// ---- POUs/AFL extensions/analog_actuator/commands/analog_actuator_deactivate.TcPOU
(*$
	Sends a deactivation command to the instance <b><i>this</i></b>, i.e.
	requests the instance to deactivate the linked <a href="#digital_output_object"><i>digital_output</i></a> <br/>	
	to reach the status <a href="#analog_actuator_status_enum"><i>ANALOG_ACTUATOR_STATUS_INACTIVE</i></a>
	The command is accepted only in <a href="#mode_enum"><i>MODE_OPERATIONAL</i></a>, the object is not faulted
	and the fault reaction is <a href="#analog_actuator_fault_reaction_enum"><i>ANALOG_ACTUATOR_FAULT_REACTION_IGNORE</i></a>.<br/>
	The method returns <i>TRUE</i> if the command is accepted, otherwise it returns <i>FALSE</i>.
$*)
FUNCTION analog_actuator_deactivate : BOOL
VAR_IN_OUT
    CONVERSION_this:	analog_actuator;	(*$ Instance to which the method applies $*)
END_VAR

IF	NOT (descriptor_mode_is_operational(CONVERSION_this.descriptor)
		OR
		descriptor_mode_is_test(CONVERSION_this.descriptor))
	OR	(
			(	descriptor_is_not_ready(CONVERSION_this.descriptor)
				AND
				CONVERSION_this.fault_reaction <> ANALOG_ACTUATOR_FAULT_REACTION_IGNORE	)
		)
THEN
	analog_actuator_deactivate := FALSE;					(* command rejected *)
 	RETURN;
END_IF

CONVERSION_this.operational_command := ANALOG_ACTUATOR_CMD_DEACTIVATE;
CONVERSION_this.analog_physical_command := 0;
analog_actuator_deactivate := TRUE;						(* command accepted *)

END_FUNCTION

// ---- POUs/AFL extensions/analog_actuator/commands/analog_actuator_set_feedback_tolerance.TcPOU
(*$
	Set Lower and Upper Feedback tolerance to the instance <b><i>this</i></b>,
	The command is accepted only in <a href="#mode_enum"><i>MODE_OPERATIONAL</i></a>
	and analog_actuator_add_ai_feedback has been called at startup
	The method returns <i>TRUE</i> if the command is accepted, otherwise it returns <i>FALSE</i>.
$*)
FUNCTION analog_actuator_set_feedback_tolerance : BOOL
VAR_INPUT
	feedback_upper_tolerance:		REAL;			(*$ Upper Tolerance Physical Value $*)
	feedback_lower_tolerance:		REAL;			(*$ Lower Tolerance Physical Value $*)
END_VAR
VAR_IN_OUT
    CONVERSION_this:	analog_actuator;	(*$ Instance to which the method applies $*)
END_VAR

IF	NOT (descriptor_mode_is_operational(CONVERSION_this.descriptor)
		OR
		descriptor_mode_is_test(CONVERSION_this.descriptor))
	OR
	NOT CONVERSION_this.has_ai_feedback
THEN
	analog_actuator_set_feedback_tolerance := FALSE;					(* command rejected *)
 	RETURN;
END_IF

CONVERSION_this.feedback_lower_tolerance := feedback_lower_tolerance;
CONVERSION_this.feedback_upper_tolerance := feedback_upper_tolerance;

analog_actuator_set_feedback_tolerance := TRUE;						(* command accepted *)

END_FUNCTION

// ---- POUs/AFL extensions/analog_actuator/initialize/analog_actuator_add_ai_feedback.TcPOU
(*$
	The method adds the <a href="#analog_input_object"><i>analog_input</i></a> that performs 
	the active feedback to the instance specified by the parameter <i><b>this</b></i>.<br/>
	<p>
	This function should be called at startup only.<br/>	
	Against errors on the input parameters the cpu is stopped, in this case the cause <br/>
	can be inspected in the global struct <i>framework.abort_error</i>: <br/>
	<br/>
	<ul>
    <li> ERRORID_1 = 9: <b><i>this</i></b> instance has already an active digital_input </li>
    <li> ERRORID_1 = 12: <b><i>this</i></b> instance is a real value check type </li>
	</ul>
	</p>
$*)
FUNCTION analog_actuator_add_ai_feedback : VOID
VAR_INPUT
	achk_diagnosis_max_value:		REAL;
	(*$ Value over which auto-diagnosis message is triggered; $*)
	achk_diagnosis_min_value:		REAL;
	(*$ Value under which auto-diagnosis message is triggered; $*)
	achk_offset:					REAL;
	(*$ Offset added (subtracted if polarity_direct is FALSE) to the other limits.
		Ex. if offset = 0 and max_value =100, out_of_upper_range is triggered if value>100
		if offset = 10 and max_value =100, out_of_upper_range is triggered if value>110 $*)
	achk_hysteresis:				UDINT;
	(*$ Hysteresis on max or min value. If max value is reached, 
		the related message can be reset only if the measured signal goes down below 
		(max value - (max value-min value)*hysteresis/100). The same for min value.; $*)
	achk_filter_on_max_value:	UDINT;
								(*$ Filter on max level reached; $*)
	achk_filter_on_min_value:	UDINT;
								(*$ Filter on min level reached; $*)
END_VAR
VAR_IN_OUT
	ai:				analog_input;
	(*$ <a href="#analog_input_object"><i>Analog_input</i></a> that has to be added $*)
	process:		process;			(*$ <a href="#process_object"><i>process</i></a> membership $*)
	CONVERSION_this:			analog_actuator;	(*$ Instance to which the method applies $*)
END_VAR

IF analog_actuator_is_not_initialized(CONVERSION_this)
   OR
   analog_input_is_not_initialized(ai)
THEN
	IF framework_initialization()
	THEN
		RETURN;
	END_IF
END_IF

IF analog_actuator_is_not_initialized(CONVERSION_this)
THEN
	framework_object_not_initialized_get_name(
		object_address := ADR(CONVERSION_this), 
		object_size := SIZEOF(CONVERSION_this), 
		abort := TRUE,
		error_str_1 := 'object not initialized',
		error_str_2 := 'analog_actuator_add_ai_feedback'
	);
    RETURN;
END_IF

IF analog_input_is_not_initialized(ai)
THEN
	framework_object_not_initialized_get_name(
		object_address := ADR(ai), 
		object_size := SIZEOF(ai),
		abort := TRUE,
		error_str_1 := 'object not initialized', 
		error_str_2 := CONCAT('Please check analog_actuator_add_ai_feedback of ',CONVERSION_this.object_name)
	);
    RETURN;
END_IF


IF (CONVERSION_this.ai_feedback<>NULL
	AND
	CONVERSION_this.ai_feedback<>ADR(ai))
THEN
	abort(
		object_name := CONVERSION_this.object_name,
		errorID_1 := 9,
		errorID_2 := 0,
		errorID_3 := 0,
		error_str_1 := CONCAT(CONVERSION_this.object_name, ' ai already used'),
		error_str_2 := ''
		);
    RETURN;
END_IF

CONVERSION_this.ai_feedback := ADR(ai);
CONVERSION_this.has_ai_feedback := TRUE;

(* todo: to define how to init analog check*)
analog_check_init(
	object_name 		:= CONCAT(CONVERSION_this.object_name,'_feedback_achk'),
	enabled_at_powerup 	:= TRUE,
	signal_type 		:= ANALOG_CHECK_PHYSICAL_VALUE,
	polarity_direct 	:= TRUE,
	diagnosis_max_value := achk_diagnosis_max_value,
	max_value 			:= achk_diagnosis_max_value,
	min_value 			:= achk_diagnosis_min_value,
	diagnosis_min_value := achk_diagnosis_min_value,
	offset 				:= achk_offset,
	hysteresis 			:= achk_hysteresis,
	filter_on_max_value := achk_filter_on_max_value,
	filter_on_min_value := achk_filter_on_min_value,
	process 			:= process,
	CONVERSION_this				:= CONVERSION_this.feedback_achk);

analog_check_add_ai(
	ai 					:= ai,
	CONVERSION_this 				:= CONVERSION_this.feedback_achk);

END_FUNCTION

// ---- POUs/AFL extensions/analog_actuator/initialize/analog_actuator_add_di_active.TcPOU
(*$
	Adds the <a href="#digital_input_object"><i>digital_input</i></a> that performs 
	the active feedback to the instance specified by the parameter <i><b>this</i></b>.
	This method must to be called only if type of analog_actuator object is <a href="#analog_actuator_type_enum"><i>ANALOG_ACTUATOR_TYPE_IN_AI</i></a> or 
	<a href="#analog_actuator_type_enum"><i>ANALOG_ACTUATOR_TYPE_IN_Ax</i></a>.<br/><br/>
	<p>
	This function should be called at startup only.<br/>	
	Against errors on the input parameters the cpu is stopped, in this case the cause <br/>
	can be inspected in the global struct <i>framework.abort_error</i>: <br/>
	<br/>
    <li> <b>ERRORID_1 = 2</b>: <b><i>this</i></b> instance has already an active digital_input </li>
    <li> <b>ERRORID_1 = 3</b>: <b><i>this</i></b> instance type doesn't allow active feedback. See 
		<a href="#analog_actuator_type_enum"><i>analog_actuator_type_enum</i></a>
	</li>
	</p>
$*)
FUNCTION analog_actuator_add_di_active: VOID
VAR_INPUT
	dchk_alarm_delay:			DINT;
	(*$ timeout (in ms) for alarm input level: when input is in alarm level for a time that exceeds this parameter then alarm on;
	if a zero value is assigned then alarm goes on immediately when the input is in alarm level $*)
END_VAR
VAR_IN_OUT
	di_active:	digital_input;
	(*$ Active <a href="#digital_input_object"><i>digital_input</i></a> that has to be added $*)
	process:	process;			(*$ <a href="#process_object"><i>process</i></a> membership $*)
	CONVERSION_this:		analog_actuator;	(*$ Instance to which the method applies $*)
END_VAR

IF CONVERSION_this.has_di_active
   AND
   CONVERSION_this.di_active = ADR(di_active)
THEN
	RETURN;
END_IF

IF analog_actuator_is_not_initialized(CONVERSION_this)
   OR
   digital_input_is_not_initialized(di_active)
THEN
	IF framework_initialization()
	THEN
		RETURN;
	END_IF
END_IF

IF analog_actuator_is_not_initialized(CONVERSION_this)
THEN
	framework_object_not_initialized_get_name(
		object_address := ADR(CONVERSION_this), 
		object_size := SIZEOF(CONVERSION_this),
		abort := TRUE,
		error_str_1 := 'object not initialized', 
		error_str_2 := 'analog_actuator_add_di_active'
	);
    RETURN;
END_IF

IF digital_input_is_not_initialized(di_active)
THEN
	framework_object_not_initialized_get_name(
		object_address := ADR(di_active), 
		object_size := SIZEOF(di_active),
		abort := TRUE, 
		error_str_1 := 'object not initialized', 
		error_str_2 := CONCAT('Please check analog_actuator_add_di_active of ',CONVERSION_this.object_name)				
	);
    RETURN;
END_IF

IF CONVERSION_this.has_di_active
   AND
   CONVERSION_this.di_active <> ADR(di_active)
THEN
    abort(
		object_name := CONVERSION_this.object_name,
        errorID_1 := 2,
        errorID_2 := 0,
        errorID_3 := 0,
        error_str_1 := CONCAT(CONVERSION_this.object_name, ' analog_actuator has already an active digital_input'),
		error_str_2 := 'analog_actuator_add_di_active'
        );
    RETURN;
END_IF

CONVERSION_this.di_active := ADR(di_active);
CONVERSION_this.has_di_active := TRUE;

digital_check_init(
	object_name			:= CONCAT(CONVERSION_this.object_name, '_active_dchk'),
	alarm_if_input_off	:= TRUE,
	alarm_delay			:= dchk_alarm_delay,
	enabled_at_powerup	:= FALSE,
	process				:= process,
	CONVERSION_this				:= CONVERSION_this.active_dchk);

digital_check_init(
	object_name			:= CONCAT(CONVERSION_this.object_name, '_inactive_dchk'),
	alarm_if_input_off	:= FALSE,
	alarm_delay			:= dchk_alarm_delay,
	enabled_at_powerup	:= FALSE,
	process				:= process,
	CONVERSION_this				:= CONVERSION_this.inactive_dchk);

digital_check_add_di(
	di					:= di_active,
	CONVERSION_this				:= CONVERSION_this.active_dchk);

digital_check_add_di(
	di					:= di_active,
	CONVERSION_this				:= CONVERSION_this.inactive_dchk);

END_FUNCTION

// ---- POUs/AFL extensions/analog_actuator/initialize/analog_actuator_add_di_ready.TcPOU
(*$
	Adds the <a href="#digital_input_object"><i>digital_input</i></a> that performs 
	the ready feedback to the instance specified by the parameter <i><b>this</i></b>.
	This method must to be called only if type of analog_actuator object is <a href="#analog_actuator_type_enum"><i>ANALOG_ACTUATOR_TYPE_IN_AI</i></a> or 
	<a href="#analog_actuator_type_enum"><i>ANALOG_ACTUATOR_TYPE_IN_Ax</i></a>.<br/><br/>
	<p>
	This function should be called at startup only.<br/>	
	Against errors on the input parameters the cpu is stopped, in this case the cause <br/>
	can be inspected in the global struct <i>framework.abort_error</i>: <br/>
	<br/>
    <li> <b>ERRORID_1 = 2</b>: <b><i>this</i></b> instance has already an active digital_input </li>
    <li> <b>ERRORID_1 = 3</b>: <b><i>this</i></b> instance type doesn't allow active feedback. See 
		<a href="#analog_actuator_type_enum"><i>analog_actuator_type_enum</i></a>
	</li>
	</p>
$*)
FUNCTION analog_actuator_add_di_ready: VOID
VAR_INPUT
	dchk_alarm_delay:			DINT;
	(*$ timeout (in ms) for alarm input level: when input is in alarm level for a time that exceeds this parameter then alarm on;
	if a zero value is assigned then alarm goes on immediately when the input is in alarm level $*)
END_VAR
VAR_IN_OUT
	di_ready:	digital_input;
	(*$ Active <a href="#digital_input_object"><i>digital_input</i></a> that has to be added $*)
	process:	process;			(*$ <a href="#process_object"><i>process</i></a> membership $*)
	CONVERSION_this:		analog_actuator;	(*$ Instance to which the method applies $*)
END_VAR

IF CONVERSION_this.has_di_ready
   AND
   CONVERSION_this.di_ready = ADR(di_ready)
THEN
	RETURN;
END_IF

IF analog_actuator_is_not_initialized(CONVERSION_this)
   OR
   digital_input_is_not_initialized(di_ready)
THEN
	IF framework_initialization()
	THEN
		RETURN;
	END_IF
END_IF

IF analog_actuator_is_not_initialized(CONVERSION_this)
THEN
	framework_object_not_initialized_get_name(
		object_address := ADR(CONVERSION_this), 
		object_size := SIZEOF(CONVERSION_this), 
		abort := TRUE,
		error_str_1 := 'object not initialized', 
		error_str_2 := 'analog_actuator_add_di_ready'
	);
    RETURN;
END_IF

IF digital_input_is_not_initialized(di_ready)
THEN
	framework_object_not_initialized_get_name(
		object_address := ADR(di_ready), 
		object_size := SIZEOF(di_ready),
		abort := TRUE, 
		error_str_1 := 'object not initialized', 
		error_str_2 := CONCAT('Please check analog_actuator_add_di_ready of ',CONVERSION_this.object_name)				
	);
    RETURN;
END_IF

IF CONVERSION_this.has_di_ready
   AND
   CONVERSION_this.di_ready <> ADR(di_ready)
THEN
    abort(
		object_name := CONVERSION_this.object_name,
        errorID_1 := 2,
        errorID_2 := 0,
        errorID_3 := 0,
        error_str_1 := CONCAT(CONVERSION_this.object_name, ' analog_actuator has already an ready digital_input'),
		error_str_2 := 'analog_actuator_add_di_ready'
        );
    RETURN;
END_IF

CONVERSION_this.di_ready := ADR(di_ready);
CONVERSION_this.has_di_ready := TRUE;

digital_check_init(
	object_name			:= CONCAT(CONVERSION_this.object_name, '_ready_dchk'),
	alarm_if_input_off	:= TRUE,
	alarm_delay			:= dchk_alarm_delay,
	enabled_at_powerup	:= FALSE,
	process				:= process,
	CONVERSION_this				:= CONVERSION_this.ready_dchk);

digital_check_add_di(
	di					:= di_ready,
	CONVERSION_this				:= CONVERSION_this.ready_dchk);

END_FUNCTION

// ---- POUs/AFL extensions/analog_actuator/initialize/analog_actuator_add_dout_activate.TcPOU
(*$
    The method adds the <a href="#digital_output_object"><i>digital_output</i></a> that performs
    the "lamp" functioning to the instance specified by the parameter <a href="#button "><i>this</i></a>.<br/>

    <p>
    This function should be called at startup only.<br/>
    Against errors on the input parameters the cpu is stopped, in this case the cause <br/>
    can be inspected in the global struct <i>framework.abort_error</i>: <br/>
    <br/>
    <li> <b>ERRORID_1 = 5</b>: <b><i>this</i></b> instance has already a digital_output </li>
    <li> <b>ERRORID_1 = 7</b>: <b><i>this</i></b> instance has already a multicolor lamp </li>
    </p>
$*)
FUNCTION analog_actuator_add_dout_activate: VOID
VAR_IN_OUT
    do_activate:   digital_output;
    (*$ Active <a href="#digital_output_object"><i>digital_output</i></a> that has to be added $*)
    CONVERSION_this:   analog_actuator; (*$ Instance to which the method applies $*)
END_VAR

IF CONVERSION_this.has_do_activate
   AND
   CONVERSION_this.do_activate = ADR(do_activate)
THEN
	RETURN;
END_IF

IF analog_actuator_is_not_initialized(CONVERSION_this)
   OR
   digital_output_is_not_initialized(do_activate)
THEN
	IF framework_initialization()
	THEN
		RETURN;
	END_IF
END_IF

IF analog_actuator_is_not_initialized(CONVERSION_this)
THEN
	framework_object_not_initialized_get_name(
		object_address := ADR(CONVERSION_this),
		object_size := SIZEOF(CONVERSION_this), 
		abort := TRUE,
		error_str_1 := 'object not initialized', 
		error_str_2 := 'analog_actuator_add_do_activate'
	);
    RETURN;
END_IF

IF digital_output_is_not_initialized(do_activate)
THEN
	framework_object_not_initialized_get_name(
		object_address := ADR(do_activate), 
		object_size := SIZEOF(do_activate),
		abort := TRUE, 
		error_str_1 := 'object not initialized',
		error_str_2 := CONCAT('Please check analog_actuator_add_do_activate of ',CONVERSION_this.object_name)				
	);
    RETURN;
END_IF

IF CONVERSION_this.has_do_activate
   AND
   CONVERSION_this.do_activate <> ADR(do_activate)
THEN
    abort(
		object_name := CONVERSION_this.object_name,
        errorID_1 := 2,
        errorID_2 := 0,
        errorID_3 := 0,
        error_str_1 := CONCAT(CONVERSION_this.object_name, ' analog_actuator has already an activate digital_output'),
		error_str_2 := 'analog_actuator_add_do_activate'
        );
    RETURN;
END_IF

CONVERSION_this.do_activate := ADR(do_activate);
CONVERSION_this.has_do_activate := TRUE;

END_FUNCTION

// ---- POUs/AFL extensions/analog_actuator/initialize/analog_actuator_init.TcPOU
(*$
	Initializes the instance specified by the parameter <b><i>this</i></b>. <br/>
	<p>
	This function should be called at startup only.<br/>	
	Against errors on the input parameters the cpu is stopped, in this case the cause <br/>
	can be inspected in the global struct <i>framework.abort_error</i>: <br/>
	<br/>
	<li> <b>ERRORID_1 = 1</b>: <b><i>object_name</i></b> is illegal </li>
	</p>
$*)
FUNCTION analog_actuator_init : VOID
VAR_INPUT
	object_name:	STRING(MAX_OBJ_NAME_LENGTH);	(*$ The instance name as <i>STRING</i> $*)
	fault_reaction:	analog_actuator_fault_reaction_enum;
													(*$ Reaction strategy in case of fault $*)
	active_time:	UDINT;
	(*$
		Activation time: see <a href="#analog_actuator_parameters"><i>active_time</i></a>
		parameter description. 
	$*)
	inactive_time:	UDINT;
	(*$
		Deactivation time: see <a href="#analog_actuator_parameters"><i>inactive_time</i></a>
		parameter description. 
	$*)
END_VAR
VAR_IN_OUT
	analog_out:		analog_output;		(*$ <a href="#analog_output_object"><i>analog_output</i></a> object to drive $*)
	process:		process;			(*$ <a href="#process_object"><i>process</i></a> membership $*)
	CONVERSION_this:			analog_actuator;	(*$ Instance to which the method applies $*)
END_VAR

IF CONVERSION_this.CONVERSION_private.initialized
THEN
	RETURN;
END_IF

IF analog_output_is_not_initialized(analog_out)
   OR
   process_is_not_initialized(process)
THEN
	IF framework_initialization()
	THEN
		RETURN;
	END_IF
END_IF

IF analog_output_is_not_initialized(analog_out)
THEN
	framework_object_not_initialized_get_name(
		object_address := ADR(analog_out),
		object_size := SIZEOF(analog_out),
		abort := TRUE,
		error_str_1 := 'object not initialized', 
		error_str_2 := CONCAT('Please check analog_actuator_init of ',CONVERSION_this.object_name)				
	);
    RETURN;
END_IF

IF process_is_not_initialized(process)
THEN
	framework_object_not_initialized_get_name(
		object_address := ADR(process), 
		object_size := SIZEOF(process), 
		abort := TRUE,
		error_str_1 := 'object not initialized', 
		error_str_2 := CONCAT('Please check analog_actuator_init of ',CONVERSION_this.object_name)			
	);
    RETURN;
END_IF

IF object_name = ''
THEN
	framework_object_not_initialized_get_name(
		object_address := ADR(CONVERSION_this), 
		object_size := SIZEOF(CONVERSION_this), 
		abort := TRUE,
		error_str_1 := 'object name is null', 
		error_str_2 := ''
	);
    RETURN;
END_IF

IF obj_name_find_illegal_characters(object_name)
THEN
    abort(
		object_name := object_name,
        errorID_1 := 1,
        errorID_2 := 0,
        errorID_3 := 0,
        error_str_1 := CONCAT(CONCAT(CONCAT(CONCAT('(', ANALOG_ACTUATOR_CLASS_NAME), ') '), object_name), ' object name is invalid'),
		error_str_2 := ''
    );
    RETURN;
END_IF

CONVERSION_this.object_name := object_name;

CONVERSION_this.CONVERSION_private.my_address := ADR(CONVERSION_this);

descriptor_init(
	object_name := CONCAT(CONVERSION_this.object_name,'.descriptor'),
	process := process,
	CONVERSION_this := CONVERSION_this.descriptor
	);

CONVERSION_this.ao_setpoint := ADR(analog_out);
analog_output_percent_write(0, analog_out);

CONVERSION_this.fault_reaction := fault_reaction;
CONVERSION_this.active_time := active_time;
CONVERSION_this.inactive_time := inactive_time;

CONVERSION_this.is_active := FALSE;
CONVERSION_this.is_inactive := FALSE;

timer_init(
	object_name := CONCAT(CONVERSION_this.object_name,'.timer'),
	process := process,
	CONVERSION_this := CONVERSION_this.timer
);

CONVERSION_this.status := ANALOG_ACTUATOR_STATUS_INIT;
CONVERSION_this.command := ANALOG_ACTUATOR_CMD_INIT;
CONVERSION_this.test.command := ANALOG_ACTUATOR_TEST_CMD_IDLE;

analog_actuator_init_snapshot(
	message_name := 'inactive_fem',
    behaviour :=  MESSAGE_BEHAVIOUR_EVENT,
	reset_timeout := 0,
	disableable := FALSE,
	individual_reset := FALSE,
	machine_reaction := MACHINE_REACTION_NORMAL_STOP,
	typology := MESSAGE_TYPOLOGY_ABNORMAL,
    analog_actuator := CONVERSION_this,
	CONVERSION_this := CONVERSION_this.inactive_fem
);

analog_actuator_init_snapshot(
	message_name := 'active_fem',
    behaviour :=  MESSAGE_BEHAVIOUR_EVENT,
	reset_timeout := 0,
	disableable := FALSE,
	individual_reset := FALSE,
	machine_reaction := MACHINE_REACTION_NORMAL_STOP,
	typology := MESSAGE_TYPOLOGY_ABNORMAL,
	analog_actuator := CONVERSION_this,
	CONVERSION_this := CONVERSION_this.active_fem
);

analog_actuator_init_snapshot(
	message_name := 'out_of_lower_range_fem',
    behaviour :=  MESSAGE_BEHAVIOUR_EVENT,
	reset_timeout := 0,
	disableable := FALSE,
	individual_reset := FALSE,
	machine_reaction := MACHINE_REACTION_NORMAL_STOP,
	typology := MESSAGE_TYPOLOGY_ABNORMAL,
    analog_actuator := CONVERSION_this,
	CONVERSION_this := CONVERSION_this.out_of_lower_range_fem
);

CONVERSION_this.CONVERSION_private.initialized := TRUE;

END_FUNCTION

// ---- POUs/AFL extensions/analog_actuator/private/analog_actuator_init_snapshot.TcPOU
(*	Inizializes a analog_actuator snapshot *)
FUNCTION analog_actuator_init_snapshot : VOID
VAR_INPUT
	message_name:		STRING(MAX_OBJ_NAME_LENGTH);(* Message name *)
	behaviour:			message_behaviour_enum;		(* Message type.
														State or event *)
    reset_timeout:      UDINT;                      (* Timeout of reset attempt valid for messages
                                                       with <a href="#message_behaviour_enum"><i>behaviour</i></a>
                                                       = MESSAGE_BEHAVIOUR_TRY_AND_CHECK *)
	disableable:		BOOL;						(* Indicates the possibility
														disable the message
														by HMI *)
	individual_reset:	BOOL;						(* Need explicit reset by
														HMI for acknowlege the message.
														TRUE = individual_reset *)
	machine_reaction:	machine_reaction_enum;		(* Machine stop type.
														(emergency, normal,	on phase, ...) *)
	typology:			message_typology_enum;		(* <a href="#message_typology_enum"><i>typology</i></a> *)
END_VAR
VAR_IN_OUT
    analog_actuator:	analog_actuator;			(* analog_actuator reference *)
	CONVERSION_this: 				analog_actuator_snapshot;	(* snapshot object reference *)
END_VAR

message_init(
    object_name := analog_actuator.object_name,
	message_name := message_name,
	owner := ADR(analog_actuator),
    behaviour :=  behaviour,
	reset_timeout := reset_timeout,
	disableable := disableable,
	individual_reset := individual_reset,
	machine_reaction := machine_reaction,
	typology := typology,
    descriptor := analog_actuator.descriptor,
	CONVERSION_this := CONVERSION_this.message
    );

CONVERSION_this.status := analog_actuator.status;
CONVERSION_this.command := analog_actuator.command;
CONVERSION_this.is_active := analog_actuator.is_active;
CONVERSION_this.is_inactive := analog_actuator.is_inactive;

END_FUNCTION

// ---- POUs/AFL extensions/analog_actuator/status/analog_actuator_get_mode.TcPOU
(*$
	Returns the current <a href="#mode_enum"><i>mode</i></a> of the instance <b><i>this</i></b>.
$*)
FUNCTION analog_actuator_get_mode: mode_enum
VAR_IN_OUT
    CONVERSION_this:	analog_actuator;	(*$ Instance to which the method applies $*)
END_VAR

analog_actuator_get_mode := descriptor_get_mode(CONVERSION_this.descriptor);

END_FUNCTION

// ---- POUs/AFL extensions/analog_actuator/status/analog_actuator_is_faulted.TcPOU
(*$
	Returns <i>TRUE</i> if the instance <b><i>this</i></b> has a fault 
	<a href="#analog_actuator_snapshot"><i>message</i></a>
    active, <i>FALSE</i> otherwise. 
$*)
FUNCTION analog_actuator_is_faulted : BOOL
VAR_IN_OUT
    CONVERSION_this:	analog_actuator;	(*$ Instance to which the method applies $*)
END_VAR

analog_actuator_is_faulted := descriptor_is_not_ready(CONVERSION_this.descriptor);

END_FUNCTION

// ---- POUs/AFL extensions/analog_actuator/status/analog_actuator_is_in_range.TcPOU
(*$
	Returns <i>TRUE</i> if the status of the instance <b><i>this</i></b> is
	<a href="#analog_actuator_status_enum"><i>ANALOG_ACTUATOR_STATUS_INACTIVE</i></a>, 
	<i>FALSE</i> otherwise.
$*)
FUNCTION analog_actuator_is_in_range: BOOL
VAR_IN_OUT
    CONVERSION_this:	analog_actuator;	(*$ Instance to which the method applies $*)
END_VAR

IF descriptor_get_mode(CONVERSION_this.descriptor) = MODE_ABSENT
THEN
	analog_actuator_is_in_range := TRUE;
	RETURN;
END_IF

analog_actuator_is_in_range := analog_check_is_in_range(CONVERSION_this.feedback_achk);

END_FUNCTION

// ---- POUs/AFL extensions/analog_actuator/status/analog_actuator_is_ready.TcPOU
(*$
	Returns <i>TRUE</i> if the status of the instance <b><i>this</i></b> is
	<a href="#analog_actuator_status_enum"><i>ANALOG_ACTUATOR_STATUS_ACTIVE</i></a>, 
	<i>FALSE</i> otherwise.
$*)
FUNCTION analog_actuator_is_ready : BOOL
VAR_IN_OUT
    CONVERSION_this:	analog_actuator;	(*$ Instance to which the method applies $*)
END_VAR

IF CONVERSION_this.has_di_ready
THEN
	analog_actuator_is_ready := digital_check_is_ready(CONVERSION_this.ready_dchk)
								AND
								descriptor_is_ready(CONVERSION_this.descriptor);
ELSE
	analog_actuator_is_ready := descriptor_is_ready(CONVERSION_this.descriptor);
END_IF

END_FUNCTION

// ---- POUs/AFL extensions/IO_Link/FUN/iol_slave_bsp00ue_configure.TcPOU

(*$
<p>This function configures a generic <a target="_blank" href="#iol_slave">iol_slave</a> as a <strong>Balluff BSP00UE</strong>. It allow to connect the object to the device-specific
parameters structure variable <a target="_blank" href="#iol_slave_bsp00ue_data">iol_slave_bsp00ue_data</a>.</p>
<p>This function should be called at startup only.</p>
$*)

FUNCTION iol_slave_bsp00ue_configure : VOID
VAR_IN_OUT
	data:						iol_slave_bsp00ue_data;			(*$	Parameters struct variable	$*)
	CONVERSION_this:			iol_slave;						(*$ Instance to which the method applies $*)
END_VAR

VAR CONSTANT
	NULL:                                   			XWORD := 0;
END_VAR

IF iol_slave_is_not_initialized(CONVERSION_this := CONVERSION_this)
	OR
	iol_slave_is_configured(CONVERSION_this := CONVERSION_this)
THEN
	RETURN;
END_IF

(*** Start parameter configuration ***)

(* STANDARD PARAMETERS CONFIGURATION *)

iol_slave_configure_parameter(
	current_value_address := ADR(CONVERSION_this.vendor_name),
	configured_value_address := NULL,
	length := SIZEOF(CONVERSION_this.vendor_name),
	_type := ADST_STRING,
	coe_index := 16#0010,
	coe_sub_index := 16#00,
	readable := TRUE,
	writeable := FALSE,
	to_check := FALSE,
	CONVERSION_this := CONVERSION_this);


iol_slave_configure_parameter(
	current_value_address := ADR(CONVERSION_this.product_name),
	configured_value_address := NULL,
	length := SIZEOF(CONVERSION_this.product_name),
	_type := ADST_STRING,
	coe_index := 16#0012,
	coe_sub_index := 16#00,
	readable := TRUE,
	writeable := FALSE,
	to_check := FALSE,
	CONVERSION_this := CONVERSION_this);

iol_slave_configure_parameter(
	current_value_address := ADR(CONVERSION_this.product_id),
	configured_value_address := NULL,
	length := SIZEOF(CONVERSION_this.product_id),
	_type := ADST_STRING,
	coe_index := 16#0013,
	coe_sub_index := 16#00,
	readable := TRUE,
	writeable := FALSE,
	to_check := FALSE,
	CONVERSION_this := CONVERSION_this);


iol_slave_configure_parameter(
	current_value_address := ADR(CONVERSION_this.hardware_revision),
	configured_value_address := NULL,
	length := SIZEOF(CONVERSION_this.hardware_revision),
	_type := ADST_STRING,
	coe_index := 16#0016,
	coe_sub_index := 16#00,
	readable := TRUE,
	writeable := FALSE,
	to_check := FALSE,
	CONVERSION_this := CONVERSION_this);

iol_slave_configure_parameter(
	current_value_address := ADR(CONVERSION_this.firmware_revision),
	configured_value_address := NULL,
	length := SIZEOF(CONVERSION_this.firmware_revision),
	_type := ADST_STRING,
	coe_index := 16#0017,
	coe_sub_index := 16#00,
	readable := TRUE,
	writeable := FALSE,
	to_check := FALSE,
	CONVERSION_this := CONVERSION_this);

iol_slave_configure_parameter(
	current_value_address := ADR(CONVERSION_this.current_app_specific_tag),
	configured_value_address := ADR(CONVERSION_this.configured_app_specific_tag),
	length := SIZEOF(CONVERSION_this.current_app_specific_tag),
	_type := ADST_STRING,
	coe_index := 16#0018,
	coe_sub_index := 16#00,
	readable := TRUE,
	writeable := TRUE,
	to_check := TRUE,
	CONVERSION_this := CONVERSION_this);

(* CUSTOM PARAMETERS CONFIGURATION *)

iol_slave_configure_parameter(
	current_value_address := ADR(data.setpoint),
	configured_value_address := NULL,
	length := SIZEOF(data.setpoint),
	_type := ADST_UINT32,
	coe_index := 60,
	coe_sub_index := 16#00,
	readable := TRUE,
	writeable := FALSE,
	to_check := FALSE,
	CONVERSION_this := CONVERSION_this);

iol_slave_configure_parameter(
	current_value_address := ADR(data.switchpoint),
	configured_value_address := NULL,
	length := SIZEOF(data.switchpoint),
	_type := ADST_UINT32,
	coe_index := 61,
	coe_sub_index := 16#00,
	readable := TRUE,
	writeable := FALSE,
	to_check := FALSE,
	CONVERSION_this := CONVERSION_this);

iol_slave_configure_parameter(
	current_value_address := ADR(data.measure_unit),
	configured_value_address := NULL,
	length := SIZEOF(data.measure_unit),
	_type := ADST_UINT8,
	coe_index := 212,
	coe_sub_index := 16#00,
	readable := TRUE,
	writeable := FALSE,
	to_check := FALSE,
	CONVERSION_this := CONVERSION_this);


iol_slave_configure_parameter(
	current_value_address := ADR(data.max_press),
	configured_value_address := NULL,
	length := SIZEOF(data.max_press),
	_type := ADST_UINT16,
	coe_index := 214,
	coe_sub_index := 16#00,
	readable := TRUE,
	writeable := FALSE,
	to_check := FALSE,
	CONVERSION_this := CONVERSION_this);


iol_slave_configure_parameter(
	current_value_address := ADR(data.min_press),
	configured_value_address := NULL,
	length := SIZEOF(data.min_press),
	_type := ADST_UINT16,
	coe_index := 213,
	coe_sub_index := 16#00,
	readable := TRUE,
	writeable := FALSE,
	to_check := FALSE,
	CONVERSION_this := CONVERSION_this);

iol_slave_configure_parameter(
	current_value_address := ADR(data.switchpoint_delay_on),
	configured_value_address := NULL,
	length := SIZEOF(data.switchpoint_delay_on),
	_type := ADST_UINT16,
	coe_index := 208,
	coe_sub_index := 16#00,
	readable := TRUE,
	writeable := FALSE,
	to_check := FALSE,
	CONVERSION_this := CONVERSION_this);

iol_slave_configure_parameter(
	current_value_address := ADR(data.switchpoint_delay_off),
	configured_value_address := NULL,
	length := SIZEOF(data.switchpoint_delay_off),
	_type := ADST_UINT16,
	coe_index := 209,
	coe_sub_index := 16#00,
	readable := TRUE,
	writeable := FALSE,
	to_check := FALSE,
	CONVERSION_this := CONVERSION_this);

iol_slave_configure_parameter(
	current_value_address := ADR(data.measure_damping),
	configured_value_address := NULL,
	length := SIZEOF(data.measure_damping),
	_type := ADST_UINT16,
	coe_index := 215,
	coe_sub_index := 16#00,
	readable := TRUE,
	writeable := FALSE,
	to_check := FALSE,
	CONVERSION_this := CONVERSION_this);

CONVERSION_this.CONVERSION_private.last_info_data_index := 6;

(*** End parameter configuration ***)
iol_slave_configuration_completed(
	parameters_ptr := ADR(data),
	parameters_struct_size := SIZEOF(data),
	CONVERSION_this := CONVERSION_this);

END_FUNCTION

// ---- POUs/AFL extensions/IO_Link/FUN/iol_slave_mlg2prime_configure.TcPOU


(*$
<p>This function configures a generic <a target="_blank" href="#iol_slave">iol_slave</a> as a <strong>Sick WTB2SC - 2P3244</strong>. It allow to connect the object to the device-specific
parameters structure variable <a target="_blank" href="#iol_slave_wtb2sc_data">iol_slave_wtb2sc_data</a>.</p>
<p>This function should be called at startup only.</p>
$*)

FUNCTION iol_slave_mlg2prime_configure : VOID
VAR_IN_OUT
	data:						iol_slave_mlg2prime_data;			(*$	Parameters struct variable$*)
	CONVERSION_this:						iol_slave;						(*$ Instance to which the method applies $*)
END_VAR

VAR CONSTANT
	NULL:                                   			XWORD := 0;
END_VAR

//IF iol_slave_is_not_initialized(CONVERSION_this := CONVERSION_this)
//	OR
IF	iol_slave_is_configured(CONVERSION_this := CONVERSION_this)
THEN
	RETURN;
END_IF

(*** Start parameter configuration ***)

(* STANDARD PARAMETERS CONFIGURATION *)

iol_slave_configure_parameter(
	current_value_address := ADR(CONVERSION_this.vendor_name),
	configured_value_address := NULL,
	length := SIZEOF(CONVERSION_this.vendor_name),
	_type := ADST_STRING,
	coe_index := 16#0010,
	coe_sub_index := 16#00,
	readable := TRUE,
	writeable := FALSE,
	to_check := FALSE,
	CONVERSION_this := CONVERSION_this);

iol_slave_configure_parameter(
	current_value_address := ADR(CONVERSION_this.product_name),
	configured_value_address := NULL,
	length := SIZEOF(CONVERSION_this.product_name),
	_type := ADST_STRING,
	coe_index := 16#0012,
	coe_sub_index := 16#00,
	readable := TRUE,
	writeable := FALSE,
	to_check := FALSE,
	CONVERSION_this := CONVERSION_this);

iol_slave_configure_parameter(
	current_value_address := ADR(CONVERSION_this.product_id),
	configured_value_address := NULL,
	length := SIZEOF(CONVERSION_this.product_id),
	_type := ADST_STRING,
	coe_index := 16#0013,
	coe_sub_index := 16#00,
	readable := TRUE,
	writeable := FALSE,
	to_check := FALSE,
	CONVERSION_this := CONVERSION_this);


iol_slave_configure_parameter(
	current_value_address := ADR(CONVERSION_this.hardware_revision),
	configured_value_address := NULL,
	length := SIZEOF(CONVERSION_this.hardware_revision),
	_type := ADST_STRING,
	coe_index := 16#0016,
	coe_sub_index := 16#00,
	readable := TRUE,
	writeable := FALSE,
	to_check := FALSE,
	CONVERSION_this := CONVERSION_this);

iol_slave_configure_parameter(
	current_value_address := ADR(CONVERSION_this.firmware_revision),
	configured_value_address := NULL,
	length := SIZEOF(CONVERSION_this.firmware_revision),
	_type := ADST_STRING,
	coe_index := 16#0017,
	coe_sub_index := 16#00,
	readable := TRUE,
	writeable := FALSE,
	to_check := FALSE,
	CONVERSION_this := CONVERSION_this);


(* CUSTOM PARAMETERS CONFIGURATION *)


iol_slave_configure_parameter(
	current_value_address := ADR(data.CrossBeamEnable),
	configured_value_address := ADR(data.CrossBeamEnable),
	length := SIZEOF(data.CrossBeamEnable),
	_type := ADST_UINT8,
	coe_index := 16#0052,
	coe_sub_index :=16#0000,
	readable := TRUE,
	writeable := TRUE,
	to_check := TRUE, (* to be evaluated *)
	CONVERSION_this := CONVERSION_this);

iol_slave_configure_parameter(
	current_value_address := ADR(data.quality_of_teach),
	configured_value_address := NULL,
	length := SIZEOF(data.quality_of_teach),
	_type := ADST_UINT8,
	coe_index := 16#00E0,
	coe_sub_index :=16#00,
	readable := TRUE,
	writeable := FALSE,
	to_check := FALSE,
	CONVERSION_this := CONVERSION_this);
	
iol_slave_configure_parameter(
	current_value_address := ADR(data.teach_result),
	configured_value_address := NULL,
	length := SIZEOF(data.teach_result),
	_type := ADST_UINT8,
	coe_index := 16#0062,
	coe_sub_index :=16#00,
	readable := TRUE,
	writeable := FALSE,
	to_check := FALSE,
	CONVERSION_this := CONVERSION_this);

iol_slave_configure_parameter(
	current_value_address := ADR(data.temperature),
	configured_value_address := NULL,
	length := SIZEOF(data.temperature),
	_type := ADST_INT8,
	coe_index := 16#0099,
	coe_sub_index :=16#00,
	readable := TRUE,
	writeable := FALSE,
	to_check := FALSE,
	CONVERSION_this := CONVERSION_this);
	
iol_slave_configure_parameter(
	current_value_address := ADR(data.quality_of_run),
	configured_value_address := NULL,
	length := SIZEOF(data.quality_of_run),
	_type := ADST_UINT8,
	coe_index := 16#00E1,
	coe_sub_index :=16#00,
	readable := TRUE,
	writeable := FALSE,
	to_check := FALSE,
	CONVERSION_this := CONVERSION_this);
	
iol_slave_configure_parameter(
	current_value_address := ADR(data.system_status),
	configured_value_address := NULL,
	length := SIZEOF(data.system_status),
	_type := ADST_UINT8,
	coe_index := 16#0064,
	coe_sub_index :=16#00,
	readable := TRUE,
	writeable := FALSE,
	to_check := FALSE,
	CONVERSION_this := CONVERSION_this);
	
iol_slave_configure_parameter(
	current_value_address := ADR(data.device_status),
	configured_value_address := NULL,
	length := SIZEOF(data.device_status),
	_type := ADST_UINT8,
	coe_index := 16#0024,
	coe_sub_index :=16#00,
	readable := TRUE,
	writeable := FALSE,
	to_check := FALSE,
	CONVERSION_this := CONVERSION_this);
	
iol_slave_configure_parameter(
	current_value_address := ADR(data.blanking_teach_enable),
	configured_value_address := ADR(data.blanking_teach_enable),
	length := SIZEOF(data.blanking_teach_enable),
	_type := ADST_UINT8,
	coe_index := 16#0046,
	coe_sub_index :=16#00,
	readable := TRUE,
	writeable := TRUE,
	to_check := TRUE,
	CONVERSION_this := CONVERSION_this);


CONVERSION_this.CONVERSION_private.last_info_data_index := 5;

(*** End parameter configuration ***)

iol_slave_configuration_completed(
	parameters_ptr := ADR(data),
	parameters_struct_size := SIZEOF(data),
	CONVERSION_this := CONVERSION_this);

END_FUNCTION

// ---- POUs/AFL extensions/jog_manager/commands/jog_manager_set_sw_limit.TcPOU
(*$
	Set sw limit value to ogject <b><i>this.axis_list[index]</i></b>.
	The method returns <i>TRUE</i> if the command is accepted, otherwise it returns <i>FALSE</i>.
$*)
FUNCTION jog_manager_set_sw_limit : BOOL
VAR_INPUT
	index:					UINT;	
	sw_limit_positive:		LREAL;
	sw_limit_negative:		LREAL;
END_VAR
VAR_IN_OUT
    CONVERSION_this:		jog_manager;	(*$ Instance to which the method applies $*)
END_VAR

IF	NOT (descriptor_mode_is_operational(CONVERSION_this.descriptor)
		(*OR
		descriptor_mode_is_test(CONVERSION_this.descriptor)*)
		OR
		(index <= JOG_MANAGER_JOG_LIST_NONE)
		OR
		(index > JOG_MANAGER_JOG_LIST_MAX))
THEN
	jog_manager_set_sw_limit := FALSE;				(* command rejected *)
 	RETURN;
END_IF

IF	CONVERSION_this.axis_list[index].axis = G_framework.NULL
THEN
	jog_manager_set_sw_limit := FALSE;				(* command rejected *)
 	RETURN;
END_IF

CONVERSION_this.axis_list[index].sw_limit_positive := sw_limit_positive;
CONVERSION_this.axis_list[index].sw_limit_negative := sw_limit_negative;
jog_manager_set_sw_limit := TRUE;						(* command accepted *)

END_FUNCTION

// ---- POUs/AFL extensions/jog_manager/private/jog_manager_init_snapshot.TcPOU
(*	Inizializes a jog_manager snapshot *)
FUNCTION jog_manager_init_snapshot : VOID
VAR_INPUT
	message_name:		STRING(MAX_OBJ_NAME_LENGTH);(* Message name *)
	behaviour:			message_behaviour_enum;		(* Message type.
														State or event *)
    reset_timeout:      UDINT;                      (* Timeout of reset attempt valid for messages
                                                       with <a href="#message_behaviour_enum"><i>behaviour</i></a>
                                                       = MESSAGE_BEHAVIOUR_TRY_AND_CHECK *)
	disableable:		BOOL;						(* Indicates the possibility
														disable the message
														by HMI *)
	individual_reset:	BOOL;						(* Need explicit reset by
														HMI for acknowlege the message.
														TRUE = individual_reset *)
	machine_reaction:	machine_reaction_enum;		(* Machine stop type.
														(emergency, normal,	on phase, ...) *)
	typology:			message_typology_enum;		(* <a href="#message_typology_enum"><i>typology</i></a> *)
END_VAR
VAR_IN_OUT
    analog_actuator:	jog_manager;			(* object reference *)
	CONVERSION_this: 	jog_manager_snapshot;	(* snapshot object reference *)
END_VAR

message_init(
    object_name := analog_actuator.object_name,
	message_name := message_name,
	owner := ADR(analog_actuator),
    behaviour :=  behaviour,
	reset_timeout := reset_timeout,
	disableable := disableable,
	individual_reset := individual_reset,
	machine_reaction := machine_reaction,
	typology := typology,
    descriptor := analog_actuator.descriptor,
	CONVERSION_this := CONVERSION_this.message);

CONVERSION_this.status := jog_manager.status;
CONVERSION_this.command := jog_manager.command;

END_FUNCTION

// ---- POUs/AFL extensions/jog_manager/private/jog_manager_set_snapshot.TcPOU
(* Dipslays a jog_manager message *)
FUNCTION jog_manager_set_snapshot : VOID
VAR_INPUT
    errorID_1:	DINT;			(* Field for specify the fault codes or enter
								   more message info *)
    errorID_2:	DINT;			(* Field for specify the fault codes or enter
								   more message info *)
    errorID_3:	DINT;			(* Field for specify the fault codes or enter
								   more message info *)
END_VAR

VAR
	owner:			POINTER TO jog_manager;
END_VAR
(*All VAR_IN_OUT variables have been moved to the end of the declaration due to compatibility reasons*)
VAR_IN_OUT
    CONVERSION_this:			jog_manager_snapshot;
								(* object snapshot reference *)
END_VAR

owner := CONVERSION_this.message.CONVERSION_private.owner;

IF message_set(errorID_1, errorID_2, errorID_3, CONVERSION_this.message)
THEN
    CONVERSION_this.status := owner^.status;
    CONVERSION_this.command := owner^.command;    
END_IF

END_FUNCTION

// ---- POUs/AFL extensions/jog_manager/status/jog_manager_get_all_slave_axis_engaged.TcPOU
(*$
	Returns <i>all_slave_axis_engaged</i> of the instance <b><i>this.axis_list[index]</i></b>.
$*)
FUNCTION jog_manager_get_all_slave_axis_engaged : BOOL
VAR_INPUT
	index:				UINT;
END_VAR
VAR_IN_OUT
    CONVERSION_this:	jog_manager;	(*$ Instance to which the method applies $*)
END_VAR

IF	(index > JOG_MANAGER_JOG_LIST_NONE)
	AND
	(index <= JOG_MANAGER_JOG_LIST_MAX)
	AND_THEN
	(CONVERSION_this.axis_list[index].axis <> G_framework.NULL)
THEN
	jog_manager_get_all_slave_axis_engaged := CONVERSION_this.axis_list[index].all_slave_axis_engaged;
ELSE
	jog_manager_get_all_slave_axis_engaged := FALSE;
END_IF

END_FUNCTION

// ---- POUs/AFL extensions/jog_manager/status/jog_manager_get_jog_activation_condition.TcPOU
(*$
	Returns <i>jog_activation_condition</i> of the instance <b><i>this</i></b>.
$*)
FUNCTION jog_manager_get_jog_activation_condition : BOOL
VAR_IN_OUT
    CONVERSION_this:	jog_manager;	(*$ Instance to which the method applies $*)
END_VAR

jog_manager_get_jog_activation_condition := CONVERSION_this.jog_activation_condition;

END_FUNCTION

// ---- POUs/AFL extensions/jog_manager/status/jog_manager_get_mode.TcPOU
(*$
	Returns the current <a href="#mode_enum"><i>mode</i></a> of the instance <b><i>this</i></b>.
$*)
FUNCTION jog_manager_get_mode: mode_enum
VAR_IN_OUT
    CONVERSION_this:	jog_manager;	(*$ Instance to which the method applies $*)
END_VAR

jog_manager_get_mode := descriptor_get_mode(CONVERSION_this.descriptor);

END_FUNCTION

// ---- POUs/AFL extensions/jog_manager/status/jog_manager_is_jog_ready.TcPOU
(*$
	Returns <i>TRUE</i> if the status of the instance <b><i>this</i></b> is
	<a href="#jog_manager_status_enum"><i>JOG_MANAGER_STATUS_READY</i></a>, 
	<i>FALSE</i> otherwise.
$*)
FUNCTION jog_manager_is_jog_ready : BOOL
VAR_IN_OUT
    CONVERSION_this:	jog_manager;	(*$ Instance to which the method applies $*)
END_VAR

jog_manager_is_jog_ready := (CONVERSION_this.status = JOG_MANAGER_STATUS_READY);

END_FUNCTION

// ---- POUs/AFL extensions/jog_manager/status/jog_manager_is_ready.TcPOU

FUNCTION jog_manager_is_ready : BOOL
VAR_IN_OUT
    CONVERSION_this:	jog_manager;	(*$ Instance to which the method applies $*)
END_VAR

IF 	CONVERSION_this.CONVERSION_private.list_selected_axis_is_valid
THEN
	jog_manager_is_ready := axis_is_ok(FALSE, CONVERSION_this.axis_list[CONVERSION_this.list_selected].axis^)
							AND
							descriptor_is_ready(CONVERSION_this.descriptor);
ELSE
	jog_manager_is_ready := descriptor_is_ready(CONVERSION_this.descriptor);
END_IF

END_FUNCTION

// ---- POUs/FB_MyQ_REAL_OOP_v2.TcPOU
FUNCTION_BLOCK FB_MyQ_REAL_OOP_v2
VAR CONSTANT
	QUEUESIZE: UDINT := 10;
END_VAR
VAR
	HoldQueue: ARRAY[1..QUEUESIZE] OF REAL;
	ProcessQueue: ARRAY[1..QUEUESIZE] OF REAL;
	Elements: UDINT;
END_VAR

METHOD M_Copy : ARRAY[1..QUEUESIZE] OF REAL
MEMCPY(ADR(M_Copy[1]), ADR(ProcessQueue[1]), SIZEOF(M_Copy));
END_METHOD

METHOD M_Insert : BOOL
VAR_INPUT
	NewValue: REAL;
END_VAR
IF Elements < QUEUESIZE THEN
	Elements := Elements + 1;
	ProcessQueue[Elements]:= NewValue;
ELSE
	Elements := QUEUESIZE;	
	MEMCPY(ADR(HoldQueue[1]), ADR(ProcessQueue[1]), SIZEOF(HoldQueue)); 
	MEMCPY(ADR(ProcessQueue[1]), ADR(HoldQueue[2]), SIZEOF(ProcessQueue)-SIZEOF(REAL));
	MEMSET(ADR(ProcessQueue[Elements]), 0, SIZEOF(REAL));
	ProcessQueue[Elements]:= NewValue;
END_IF
END_METHOD

METHOD M_Peek : REAL
IF Elements > 0 THEN
	M_Peek := ProcessQueue[1];
END_IF
END_METHOD

METHOD M_Remove : REAL
IF Elements > 0 THEN
	M_Remove := ProcessQueue[1];
	MEMCPY(ADR(HoldQueue[1]), ADR(ProcessQueue[1]), SIZEOF(HoldQueue)); 
	MEMCPY(ADR(ProcessQueue[1]), ADR(HoldQueue[2]), SIZEOF(ProcessQueue)-SIZEOF(REAL));
	MEMSET(ADR(ProcessQueue[Elements]), 0, SIZEOF(REAL));
	Elements := Elements - 1;
END_IF
END_METHOD

METHOD M_Reset : BOOL
MEMSET(ADR(HoldQueue[1]), 0, SIZEOF(HoldQueue));
MEMSET(ADR(ProcessQueue[1]), 0, SIZEOF(ProcessQueue));	
Elements := 0;
END_METHOD

PROPERTY P_Count : UDINT
GET
P_Count:=Elements;
END_GET
END_PROPERTY

PROPERTY P_FIFOSize : UDINT
GET
P_FIFOSize:=QUEUESIZE;
END_GET
END_PROPERTY

END_FUNCTION_BLOCK

// ---- Tools/Common/interface_configuration.TcPOU
FUNCTION interface_configuration : VOID
VAR_IN_OUT
	motman:																motorization_manager;
	machine:															machine;
		
	cabinet_safety_controller:											safety_integrated_controller;
	drives_safety_controller:											safety_integrated_controller;

	cabinet_ethercat_master:											net_ethercat_master;
	carton_forming_ethercat_master:										net_ethercat_master;	

	emergency_series:													safety_integrated_series;	
	delayed_emergency_series:											safety_integrated_series;

	(* Machine encoders *)
	wu_cartonPickup_drums_motorization_encoder_axis:					axis;
	wu_cartonPickup_drums_motorization_simulation_encoder_axis:			axis;
	
	wu_cartonForming_wheel_motorization_encoder_axis:					axis;
	wu_cartonForming_wheel_motorization_simulation_encoder_axis:		axis;
	
	(* Drives *)
	wu_cartonForming_wheel_motorization_drv:							soe_drive;
	wu_cartonPickup_drums_motorization_drv:								soe_drive;
	wu_cartonFeeding_leftSide_belt_drv:									soe_drive;
	wu_cartonFeeding_leftSide_hopperBelt_drv:							soe_drive;
	wu_cartonFeeding_rightSide_belt_drv:								soe_drive;
	wu_cartonFeeding_rightSide_hopperBelt_drv:							soe_drive;
	wu_cartonFeeding_presser_drv:										soe_drive;	
	wu_cupsFeeding_conveyor_drv:										soe_drive;
	wu_cupsFeeding_cochlea_drv:											soe_drive;
	wu_cupsFeeding_innerSide_belt_drv:									soe_drive;
	wu_cupsFeeding_outerSide_belt_drv:									soe_drive;	
	wu_twistedCups_conveyor_drv:										soe_drive;
	wu_cartonFilling_lowerBelts_innerPusher_drv:						soe_drive;
	wu_cartonFilling_lowerBelts_innerCounterPusher_drv:					soe_drive;	
	wu_cartonFilling_lowerBelts_outerPusher_drv:						soe_drive;	
	wu_cartonFilling_lowerBelts_outerCounterPusher_drv:					soe_drive;
	
	wu_cartonFilling_justifiers_innerPusher_drv:						soe_drive;
	wu_cartonFilling_justifiers_outerPusher_drv:						soe_drive;	
	wu_cartonFilling_justifiers_outerCounterPusher_drv:					soe_drive;	
	
	wu_main_oilLubrication_basement1_pumpRecoveryWheel_axis_drv:		soe_drive;
	wu_main_oilLubrication_recoveryPump_axis_drv:						soe_drive;
	(* Drives series *)	
	wu_cartonForming_wheel_motorization_drv_smes:						safety_integrated_series;
	wu_cartonForming_wheel_motorization_drv_smm1:						safety_integrated_series;
	
	wu_cartonPickup_drums_motorization_drv_smes:						safety_integrated_series;
	wu_cartonPickup_drums_motorization_drv_smm1:						safety_integrated_series;

	wu_cartonFeeding_leftSide_belt_drv_smes:							safety_integrated_series;
	wu_cartonFeeding_leftSide_belt_drv_smm1:							safety_integrated_series;
	
	wu_cartonFeeding_leftSide_hopperBelt_drv_smes:						safety_integrated_series;
	wu_cartonFeeding_leftSide_hopperBelt_drv_smm1:						safety_integrated_series;	

	wu_cartonFeeding_rightSide_belt_drv_smes:							safety_integrated_series;
	wu_cartonFeeding_rightSide_belt_drv_smm1:							safety_integrated_series;
	
	wu_cartonFeeding_rightSide_hopperBelt_drv_smes:						safety_integrated_series;
	wu_cartonFeeding_rightSide_hopperBelt_drv_smm1:						safety_integrated_series;	

	wu_cartonFeeding_presser_drv_smes:									safety_integrated_series;
	wu_cartonFeeding_presser_drv_smm1:									safety_integrated_series;

	wu_cupsFeeding_conveyor_drv_smes:									safety_integrated_series;
			
	wu_cupsFeeding_cochlea_drv_smes:									safety_integrated_series;
	wu_cupsFeeding_cochlea_drv_smm1:									safety_integrated_series;
	
	wu_cupsFeeding_innerSide_belt_drv_smes:								safety_integrated_series;
	wu_cupsFeeding_outerSide_belt_drv_smes:								safety_integrated_series;

	wu_twistedCups_conveyor_drv_smes:									safety_integrated_series;

	wu_cartonFilling_lowerBelts_innerPusher_drv_smes:					safety_integrated_series;
	wu_cartonFilling_lowerBelts_innerCounterPusher_drv_smes:			safety_integrated_series;	
	wu_cartonFilling_lowerBelts_outerPusher_drv_smes:					safety_integrated_series;	
	wu_cartonFilling_lowerBelts_outerCounterPusher_drv_smes:			safety_integrated_series;

	wu_cartonFilling_justifiers_innerPusher_drv_smes:					safety_integrated_series;
	wu_cartonFilling_justifiers_outerPusher_drv_smes:					safety_integrated_series;	
	wu_cartonFilling_justifiers_outerCounterPusher_drv_smes:			safety_integrated_series;
	
	wu_main_oilLubrication_basement1_pumpRecoveryWheel_axis_drv_sems:   safety_integrated_series;
	wu_main_oilLubrication_basement1_pumpRecoveryWheel_axis_drv_smm1:	safety_integrated_series;
	
	wu_main_oilLubrication_recoveryPump_axis_drv_smes:					safety_integrated_series;
	wu_main_oilLubrication_recoveryPump_axis_drv_smm1:					safety_integrated_series;
	
	CONVERSION_this:													wu_main_configurator_struct;			
END_VAR

CONVERSION_this.motman_ref																:= ADR(motman);
CONVERSION_this.machine_ref																:= ADR(machine);

CONVERSION_this.cabinet_safety_controller_ref											:= ADR(cabinet_safety_controller);
CONVERSION_this.drives_safety_controller_ref											:= ADR(drives_safety_controller);

CONVERSION_this.cabinet_ethercat_master_ref												:= ADR(cabinet_ethercat_master);
CONVERSION_this.carton_forming_ethercat_master_ref										:= ADR(carton_forming_ethercat_master);

CONVERSION_this.emergency_series_ref													:= ADR(emergency_series);
CONVERSION_this.delayed_emergency_series_ref											:= ADR(delayed_emergency_series);

(* Axis *)
IF framework_is_local_simulated()
THEN
	CONVERSION_this.drums_encoder_ref 														:= ADR(wu_cartonPickup_drums_motorization_simulation_encoder_axis);
	CONVERSION_this.wheel_encoder_ref														:= ADR(wu_cartonForming_wheel_motorization_simulation_encoder_axis);
ELSE
	CONVERSION_this.drums_encoder_ref 														:= ADR(wu_cartonPickup_drums_motorization_encoder_axis);
	CONVERSION_this.wheel_encoder_ref														:= ADR(wu_cartonForming_wheel_motorization_encoder_axis);
END_IF

CONVERSION_this.wu_main_oilLubrication_basement1_pumpRecoveryWheel_axis_drv_ref			:= ADR(wu_main_oilLubrication_basement1_pumpRecoveryWheel_axis_drv);
CONVERSION_this.wu_main_oilLubrication_basement1_pumpRecoveryWheel_axis_drv_sems_ref	:= ADR(wu_main_oilLubrication_basement1_pumpRecoveryWheel_axis_drv_sems);
CONVERSION_this.wu_main_oilLubrication_basement1_pumpRecoveryWheel_axis_drv_smm1_ref	:= ADR(wu_main_oilLubrication_basement1_pumpRecoveryWheel_axis_drv_smm1);

CONVERSION_this.wu_main_oilLubrication_recoveryPump_axis_drv_ref						:= ADR(wu_main_oilLubrication_recoveryPump_axis_drv);
CONVERSION_this.wu_main_oilLubrication_recoveryPump_axis_drv_smes_ref					:= ADR(wu_main_oilLubrication_basement1_pumpRecoveryWheel_axis_drv_sems);
CONVERSION_this.wu_main_oilLubrication_recoveryPump_axis_drv_smm1_ref					:= ADR(wu_main_oilLubrication_basement1_pumpRecoveryWheel_axis_drv_smm1);

CONVERSION_this.wu_cartonForming_wheel_motorization_drv_ref								:= ADR(wu_cartonForming_wheel_motorization_drv);
CONVERSION_this.wu_cartonForming_wheel_motorization_drv_smes_ref						:= ADR(wu_cartonForming_wheel_motorization_drv_smes);
CONVERSION_this.wu_cartonForming_wheel_motorization_drv_smm1_ref						:= ADR(wu_cartonForming_wheel_motorization_drv_smm1);

CONVERSION_this.wu_cartonPickup_drums_motorization_drv_ref								:= ADR(wu_cartonPickup_drums_motorization_drv);
CONVERSION_this.wu_cartonPickup_drums_motorization_drv_smes_ref							:= ADR(wu_cartonPickup_drums_motorization_drv_smes);
CONVERSION_this.wu_cartonPickup_drums_motorization_drv_smm1_ref							:= ADR(wu_cartonPickup_drums_motorization_drv_smm1);

CONVERSION_this.wu_cartonFeeding_leftSide_belt_drv_ref									:= ADR(wu_cartonFeeding_leftSide_belt_drv);
CONVERSION_this.wu_cartonFeeding_leftSide_belt_drv_smes_ref								:= ADR(wu_cartonFeeding_leftSide_belt_drv_smes);
CONVERSION_this.wu_cartonFeeding_leftSide_belt_drv_smm1_ref								:= ADR(wu_cartonFeeding_leftSide_belt_drv_smm1);

CONVERSION_this.wu_cartonFeeding_leftSide_hopperBelt_drv_ref							:= ADR(wu_cartonFeeding_leftSide_hopperBelt_drv);
CONVERSION_this.wu_cartonFeeding_leftSide_hopperBelt_drv_smes_ref						:= ADR(wu_cartonFeeding_leftSide_hopperBelt_drv_smes);
CONVERSION_this.wu_cartonFeeding_leftSide_hopperBelt_drv_smm1_ref						:= ADR(wu_cartonFeeding_leftSide_hopperBelt_drv_smm1);

CONVERSION_this.wu_cartonFeeding_rightSide_belt_drv_ref									:= ADR(wu_cartonFeeding_rightSide_belt_drv);
CONVERSION_this.wu_cartonFeeding_rightSide_belt_drv_smes_ref							:= ADR(wu_cartonFeeding_rightSide_belt_drv_smes);
CONVERSION_this.wu_cartonFeeding_rightSide_belt_drv_smm1_ref							:= ADR(wu_cartonFeeding_rightSide_belt_drv_smm1);

CONVERSION_this.wu_cartonFeeding_rightSide_hopperBelt_drv_ref							:= ADR(wu_cartonFeeding_rightSide_hopperBelt_drv);
CONVERSION_this.wu_cartonFeeding_rightSide_hopperBelt_drv_smes_ref						:= ADR(wu_cartonFeeding_rightSide_hopperBelt_drv_smes);
CONVERSION_this.wu_cartonFeeding_rightSide_hopperBelt_drv_smm1_ref						:= ADR(wu_cartonFeeding_rightSide_hopperBelt_drv_smm1);
	
CONVERSION_this.wu_cartonFeeding_presser_drv_ref										:= ADR(wu_cartonFeeding_presser_drv);
CONVERSION_this.wu_cartonFeeding_presser_drv_smes_ref									:= ADR(wu_cartonFeeding_presser_drv_smes);
CONVERSION_this.wu_cartonFeeding_presser_drv_smm1_ref									:= ADR(wu_cartonFeeding_presser_drv_smm1);

CONVERSION_this.wu_cupsFeeding_conveyor_drv_ref											:= ADR(wu_cupsFeeding_conveyor_drv);
CONVERSION_this.wu_cupsFeeding_conveyor_drv_smes_ref									:= ADR(wu_cupsFeeding_conveyor_drv_smes);

CONVERSION_this.wu_cupsFeeding_cochlea_drv_ref											:= ADR(wu_cupsFeeding_cochlea_drv);
CONVERSION_this.wu_cupsFeeding_cochlea_drv_smes_ref										:= ADR(wu_cupsFeeding_cochlea_drv_smes);
CONVERSION_this.wu_cupsFeeding_cochlea_drv_smm1_ref										:= ADR(wu_cupsFeeding_cochlea_drv_smm1);

CONVERSION_this.wu_cupsFeeding_innerSide_belt_drv_ref									:= ADR(wu_cupsFeeding_innerSide_belt_drv);
CONVERSION_this.wu_cupsFeeding_innerSide_belt_drv_smes_ref								:= ADR(wu_cupsFeeding_innerSide_belt_drv_smes);

CONVERSION_this.wu_cupsFeeding_outerSide_belt_drv_ref									:= ADR(wu_cupsFeeding_outerSide_belt_drv);
CONVERSION_this.wu_cupsFeeding_outerSide_belt_drv_smes_ref								:= ADR(wu_cupsFeeding_outerSide_belt_drv_smes);

CONVERSION_this.wu_twistedCups_conveyor_drv_ref											:= ADR(wu_twistedCups_conveyor_drv);
CONVERSION_this.wu_twistedCups_conveyor_drv_smes_ref									:= ADR(wu_twistedCups_conveyor_drv_smes);

CONVERSION_this.wu_cartonFilling_lowerBelts_innerPusher_drv_ref							:= ADR(wu_cartonFilling_lowerBelts_innerPusher_drv);
CONVERSION_this.wu_cartonFilling_lowerBelts_innerPusher_drv_smes_ref					:= ADR(wu_cartonFilling_lowerBelts_innerPusher_drv_smes);

CONVERSION_this.wu_cartonFilling_lowerBelts_innerCounterPusher_drv_ref					:= ADR(wu_cartonFilling_lowerBelts_innerCounterPusher_drv);
CONVERSION_this.wu_cartonFilling_lowerBelts_innerCounterPusher_drv_smes_ref				:= ADR(wu_cartonFilling_lowerBelts_innerCounterPusher_drv_smes);

CONVERSION_this.wu_cartonFilling_lowerBelts_outerPusher_drv_ref							:= ADR(wu_cartonFilling_lowerBelts_outerPusher_drv);
CONVERSION_this.wu_cartonFilling_lowerBelts_outerPusher_drv_smes_ref					:= ADR(wu_cartonFilling_lowerBelts_outerPusher_drv_smes);

CONVERSION_this.wu_cartonFilling_lowerBelts_outerCounterPusher_drv_ref					:= ADR(wu_cartonFilling_lowerBelts_outerCounterPusher_drv);
CONVERSION_this.wu_cartonFilling_lowerBelts_outerCounterPusher_drv_smes_ref				:= ADR(wu_cartonFilling_lowerBelts_outerCounterPusher_drv_smes);

CONVERSION_this.wu_cartonFilling_justifiers_innerPusher_drv_ref							:= ADR(wu_cartonFilling_justifiers_innerPusher_drv);
CONVERSION_this.wu_cartonFilling_justifiers_innerPusher_drv_smes_ref					:= ADR(wu_cartonFilling_justifiers_innerPusher_drv_smes);

CONVERSION_this.wu_cartonFilling_justifiers_outerPusher_drv_ref							:= ADR(wu_cartonFilling_justifiers_outerPusher_drv);
CONVERSION_this.wu_cartonFilling_justifiers_outerPusher_drv_smes_ref					:= ADR(wu_cartonFilling_justifiers_outerPusher_drv_smes);

CONVERSION_this.wu_cartonFilling_justifiers_outerCounterPusher_drv_ref					:= ADR(wu_cartonFilling_justifiers_outerCounterPusher_drv);
CONVERSION_this.wu_cartonFilling_justifiers_outerCounterPusher_drv_smes_ref				:= ADR(wu_cartonFilling_justifiers_outerCounterPusher_drv_smes);

END_FUNCTION

// ---- _Debug/dbg_csp_case_closing_ls_horizontal.TcPOU

(********************* G.D S.p.A. - Technical Department ***********************************
This program has been generated automatically from Application Designer DE&F
********************************************************************************************)
PROGRAM dbg_csp_case_closing_ls_horizontal
VAR
  axis_shd : axis_shadow;
END_VAR

_objects_manager();

IF	g_application_status <> APPLICATION_STATUS_RUNNING
THEN
	RETURN;
END_IF

CASE process_get_mode(CONVERSION_this := dbg_root.prc) OF
	MODE_ABSENT,
	MODE_INACTIVE:
		RETURN;
	MODE_TEST:
		RETURN;
END_CASE

ACTION _objects_manager:
IF	objects_initialization()
THEN
	axis_shadow_init(
		sim_mode:= SHADOW_SIMULATION_MODE_AUTOMATIC, 
		father:= csp_case_closing_ls_horizontal.axis, 
		process:= dbg_root.prc, 
		CONVERSION_this:= axis_shd);

	RETURN;
END_IF

IF	objects_running()
THEN
	axis_shadow_cycle(axis_shd);
END_IF
END_ACTION

END_PROGRAM

// ---- _Debug/dbg_root.TcPOU

(********************* G.D S.p.A. - Technical Department ***********************************
This program has been generated automatically from Application Designer DE&F
********************************************************************************************)
PROGRAM dbg_root
VAR
	prc:		process;
	debug_mch:	machine;
  csp_mch_shd : machine_shadow;
  dbg_root_debug_mch_shd : machine_shadow;
END_VAR

_read_var_input();
_objects_manager();

IF	g_application_status <> APPLICATION_STATUS_RUNNING
THEN
	RETURN;
END_IF

_read_process_image();
_mode_manager();

CASE process_get_mode(CONVERSION_this := prc) OF
	MODE_ABSENT,
	MODE_INACTIVE:
		RETURN;
	MODE_TEST:
		_handle_process_test();
		RETURN;
END_CASE

_set_runtime_properties();

_write_output();

ACTION _handle_process_test:
;
END_ACTION

ACTION _mode_manager:
IF	process_mode_req_is_pending(CONVERSION_this := prc)
THEN
    process_apply_mode_req_first_step(CONVERSION_this := prc);
    CASE process_get_mode(CONVERSION_this := prc) OF
        MODE_TO_ABSENT:
            ;
        MODE_TO_INACTIVE:
            ;
        MODE_TO_TEST:
            ;
        MODE_TO_OPERATIONAL:
            ;
    END_CASE
    process_apply_mode_req_second_step(CONVERSION_this := prc);
END_IF
END_ACTION

ACTION _objects_manager:
IF	objects_initialization()
THEN
	machine_init(
		object_name 	:=	'dbg_root.mch',
		name_to_hmi 	:=	'Debug',
		CONVERSION_this :=	debug_mch);

	process_init(
		object_name 	:=	'dbg_root.prc',
		machine 		:=	dbg_root.debug_mch,
		CONVERSION_this :=	prc);
	machine_shadow_init(
		sim_mode:= SHADOW_SIMULATION_MODE_AUTOMATIC, 
		father:= csp.mch, 
		process:= dbg_root.prc, 
		CONVERSION_this:= csp_mch_shd);

	machine_shadow_init(
		sim_mode:= SHADOW_SIMULATION_MODE_AUTOMATIC, 
		father:= dbg_root.debug_mch, 
		process:= dbg_root.prc, 
		CONVERSION_this:= dbg_root_debug_mch_shd);


	RETURN;
END_IF

IF	objects_running()
THEN
    process_cycle(CONVERSION_this := prc);
	machine_shadow_cycle(csp_mch_shd);
	machine_shadow_cycle(dbg_root_debug_mch_shd);
END_IF
END_ACTION

ACTION _read_process_image:
;
END_ACTION

ACTION _read_var_input:
;
END_ACTION

ACTION _set_runtime_properties:
;
END_ACTION

ACTION _write_output:
;
END_ACTION

END_PROGRAM

// ---- _Debug/dbg_csp_case_closing_ls_lower.TcPOU

(********************* G.D S.p.A. - Technical Department ***********************************
This program has been generated automatically from Application Designer DE&F
********************************************************************************************)
PROGRAM dbg_csp_case_closing_ls_lower
VAR
  axis_shd : axis_shadow;
END_VAR

_objects_manager();

IF	g_application_status <> APPLICATION_STATUS_RUNNING
THEN
	RETURN;
END_IF

CASE process_get_mode(CONVERSION_this := dbg_root.prc) OF
	MODE_ABSENT,
	MODE_INACTIVE:
		RETURN;
	MODE_TEST:
		RETURN;
END_CASE

ACTION _objects_manager:
IF	objects_initialization()
THEN
	axis_shadow_init(
		sim_mode:= SHADOW_SIMULATION_MODE_AUTOMATIC, 
		father:= csp_case_closing_ls_lower.axis, 
		process:= dbg_root.prc, 
		CONVERSION_this:= axis_shd);

	RETURN;
END_IF

IF	objects_running()
THEN
	axis_shadow_cycle(axis_shd);
END_IF
END_ACTION

END_PROGRAM

// ---- _Debug/dbg_csp_case_closing_ls_upper.TcPOU

(********************* G.D S.p.A. - Technical Department ***********************************
This program has been generated automatically from Application Designer DE&F
********************************************************************************************)
PROGRAM dbg_csp_case_closing_ls_upper
VAR
  axis_shd : axis_shadow;
END_VAR

_objects_manager();

IF	g_application_status <> APPLICATION_STATUS_RUNNING
THEN
	RETURN;
END_IF

CASE process_get_mode(CONVERSION_this := dbg_root.prc) OF
	MODE_ABSENT,
	MODE_INACTIVE:
		RETURN;
	MODE_TEST:
		RETURN;
END_CASE

ACTION _objects_manager:
IF	objects_initialization()
THEN
	axis_shadow_init(
		sim_mode:= SHADOW_SIMULATION_MODE_AUTOMATIC, 
		father:= csp_case_closing_ls_upper.axis, 
		process:= dbg_root.prc, 
		CONVERSION_this:= axis_shd);

	RETURN;
END_IF

IF	objects_running()
THEN
	axis_shadow_cycle(axis_shd);
END_IF
END_ACTION

END_PROGRAM

// ---- _Debug/dbg_csp_case_closing_os_horizontal.TcPOU

(********************* G.D S.p.A. - Technical Department ***********************************
This program has been generated automatically from Application Designer DE&F
********************************************************************************************)
PROGRAM dbg_csp_case_closing_os_horizontal
VAR
  axis_shd : axis_shadow;
END_VAR

_objects_manager();

IF	g_application_status <> APPLICATION_STATUS_RUNNING
THEN
	RETURN;
END_IF

CASE process_get_mode(CONVERSION_this := dbg_root.prc) OF
	MODE_ABSENT,
	MODE_INACTIVE:
		RETURN;
	MODE_TEST:
		RETURN;
END_CASE

ACTION _objects_manager:
IF	objects_initialization()
THEN
	axis_shadow_init(
		sim_mode:= SHADOW_SIMULATION_MODE_AUTOMATIC, 
		father:= csp_case_closing_os_horizontal.axis, 
		process:= dbg_root.prc, 
		CONVERSION_this:= axis_shd);

	RETURN;
END_IF

IF	objects_running()
THEN
	axis_shadow_cycle(axis_shd);
END_IF
END_ACTION

END_PROGRAM

// ---- _Debug/dbg_csp_case_closing_os_lower.TcPOU

(********************* G.D S.p.A. - Technical Department ***********************************
This program has been generated automatically from Application Designer DE&F
********************************************************************************************)
PROGRAM dbg_csp_case_closing_os_lower
VAR
  axis_shd : axis_shadow;
END_VAR

_objects_manager();

IF	g_application_status <> APPLICATION_STATUS_RUNNING
THEN
	RETURN;
END_IF

CASE process_get_mode(CONVERSION_this := dbg_root.prc) OF
	MODE_ABSENT,
	MODE_INACTIVE:
		RETURN;
	MODE_TEST:
		RETURN;
END_CASE

ACTION _objects_manager:
IF	objects_initialization()
THEN
	axis_shadow_init(
		sim_mode:= SHADOW_SIMULATION_MODE_AUTOMATIC, 
		father:= csp_case_closing_os_lower.axis, 
		process:= dbg_root.prc, 
		CONVERSION_this:= axis_shd);

	RETURN;
END_IF

IF	objects_running()
THEN
	axis_shadow_cycle(axis_shd);
END_IF
END_ACTION

END_PROGRAM

// ---- _Debug/dbg_csp_case_closing_os_upper.TcPOU

(********************* G.D S.p.A. - Technical Department ***********************************
This program has been generated automatically from Application Designer DE&F
********************************************************************************************)
PROGRAM dbg_csp_case_closing_os_upper
VAR
  axis_shd : axis_shadow;
END_VAR

_objects_manager();

IF	g_application_status <> APPLICATION_STATUS_RUNNING
THEN
	RETURN;
END_IF

CASE process_get_mode(CONVERSION_this := dbg_root.prc) OF
	MODE_ABSENT,
	MODE_INACTIVE:
		RETURN;
	MODE_TEST:
		RETURN;
END_CASE

ACTION _objects_manager:
IF	objects_initialization()
THEN
	axis_shadow_init(
		sim_mode:= SHADOW_SIMULATION_MODE_AUTOMATIC, 
		father:= csp_case_closing_os_upper.axis, 
		process:= dbg_root.prc, 
		CONVERSION_this:= axis_shd);

	RETURN;
END_IF

IF	objects_running()
THEN
	axis_shadow_cycle(axis_shd);
END_IF
END_ACTION

END_PROGRAM

// ---- _Debug/dbg_csp_case_discharge_accu_depth.TcPOU

(********************* G.D S.p.A. - Technical Department ***********************************
This program has been generated automatically from Application Designer DE&F
********************************************************************************************)
PROGRAM dbg_csp_case_discharge_accu_depth
VAR
  axis_shd : axis_shadow;
END_VAR

_objects_manager();

IF	g_application_status <> APPLICATION_STATUS_RUNNING
THEN
	RETURN;
END_IF

CASE process_get_mode(CONVERSION_this := dbg_root.prc) OF
	MODE_ABSENT,
	MODE_INACTIVE:
		RETURN;
	MODE_TEST:
		RETURN;
END_CASE

ACTION _objects_manager:
IF	objects_initialization()
THEN
	axis_shadow_init(
		sim_mode:= SHADOW_SIMULATION_MODE_AUTOMATIC, 
		father:= csp_case_feed_reject_accU_depth.axis, 
		process:= dbg_root.prc, 
		CONVERSION_this:= axis_shd);

	RETURN;
END_IF

IF	objects_running()
THEN
	axis_shadow_cycle(axis_shd);
END_IF
END_ACTION

END_PROGRAM

// ---- _Debug/dbg_csp_case_discharge_belts_conveyor.TcPOU

(********************* G.D S.p.A. - Technical Department ***********************************
This program has been generated automatically from Application Designer DE&F
********************************************************************************************)
PROGRAM dbg_csp_case_discharge_belts_conveyor
VAR
  axis_shd : axis_shadow;
END_VAR

_objects_manager();

IF	g_application_status <> APPLICATION_STATUS_RUNNING
THEN
	RETURN;
END_IF

CASE process_get_mode(CONVERSION_this := dbg_root.prc) OF
	MODE_ABSENT,
	MODE_INACTIVE:
		RETURN;
	MODE_TEST:
		RETURN;
END_CASE

ACTION _objects_manager:
IF	objects_initialization()
THEN
	axis_shadow_init(
		sim_mode:= SHADOW_SIMULATION_MODE_AUTOMATIC, 
		father:= csp_case_discharge_belts_conveyor.axis, 
		process:= dbg_root.prc, 
		CONVERSION_this:= axis_shd);

	RETURN;
END_IF

IF	objects_running()
THEN
	axis_shadow_cycle(axis_shd);
END_IF
END_ACTION

END_PROGRAM

// ---- _Debug/dbg_csp_case_discharge_belts_rotate.TcPOU

(********************* G.D S.p.A. - Technical Department ***********************************
This program has been generated automatically from Application Designer DE&F
********************************************************************************************)
PROGRAM dbg_csp_case_discharge_belts_rotate
VAR
  axis_shd : axis_shadow;
END_VAR

_objects_manager();

IF	g_application_status <> APPLICATION_STATUS_RUNNING
THEN
	RETURN;
END_IF

CASE process_get_mode(CONVERSION_this := dbg_root.prc) OF
	MODE_ABSENT,
	MODE_INACTIVE:
		RETURN;
	MODE_TEST:
		RETURN;
END_CASE

ACTION _objects_manager:
IF	objects_initialization()
THEN
	axis_shadow_init(
		sim_mode:= SHADOW_SIMULATION_MODE_AUTOMATIC, 
		father:= csp_case_discharge_belts_rotate.axis, 
		process:= dbg_root.prc, 
		CONVERSION_this:= axis_shd);

	RETURN;
END_IF

IF	objects_running()
THEN
	axis_shadow_cycle(axis_shd);
END_IF
END_ACTION

END_PROGRAM

// ---- _Debug/dbg_csp_case_discharge_reject_belt.TcPOU

(********************* G.D S.p.A. - Technical Department ***********************************
This program has been generated automatically from Application Designer DE&F
********************************************************************************************)
PROGRAM dbg_csp_case_discharge_reject_belt
VAR
  axis_shd : axis_shadow;
END_VAR

_objects_manager();

IF	g_application_status <> APPLICATION_STATUS_RUNNING
THEN
	RETURN;
END_IF

CASE process_get_mode(CONVERSION_this := dbg_root.prc) OF
	MODE_ABSENT,
	MODE_INACTIVE:
		RETURN;
	MODE_TEST:
		RETURN;
END_CASE

ACTION _objects_manager:
IF	objects_initialization()
THEN
	axis_shadow_init(
		sim_mode:= SHADOW_SIMULATION_MODE_AUTOMATIC, 
		father:= csp_case_discharge_reject_belt.axis, 
		process:= dbg_root.prc, 
		CONVERSION_this:= axis_shd);

	RETURN;
END_IF

IF	objects_running()
THEN
	axis_shadow_cycle(axis_shd);
END_IF
END_ACTION

END_PROGRAM

// ---- _Debug/dbg_csp_case_discharge_reject_sensors.TcPOU

(********************* G.D S.p.A. - Technical Department ***********************************
This program has been generated automatically from Application Designer DE&F
********************************************************************************************)
PROGRAM dbg_csp_case_discharge_reject_sensors
VAR
  downstream_backup_di_shd : digital_input_shadow;
  downstream_backup_di_dchk_shd : digital_check_shadow;
  reject_backup_di_shd : digital_input_shadow;
  reject_backup_di_dchk_shd : digital_check_shadow;
  reject_present_di_shd : digital_input_shadow;
  reject_present_di_dchk_shd : digital_check_shadow;
  reject_trigger_di_shd : digital_input_shadow;
  reject_trigger_inchoerence_chksect_shd : check_section_shadow;
END_VAR

_objects_manager();

IF	g_application_status <> APPLICATION_STATUS_RUNNING
THEN
	RETURN;
END_IF

CASE process_get_mode(CONVERSION_this := dbg_root.prc) OF
	MODE_ABSENT,
	MODE_INACTIVE:
		RETURN;
	MODE_TEST:
		RETURN;
END_CASE

ACTION _objects_manager:
IF	objects_initialization()
THEN
	digital_input_shadow_init(
		sim_mode:= SHADOW_SIMULATION_MODE_AUTOMATIC, 
		father:= csp_case_discharge_reject_sensors.downstream_backup_di, 
		process:= dbg_root.prc, 
		CONVERSION_this:= downstream_backup_di_shd);

	digital_check_shadow_init(
		sim_mode:= SHADOW_SIMULATION_MODE_AUTOMATIC, 
		father:= csp_case_discharge_reject_sensors.downstream_backup_di_dchk, 
		process:= dbg_root.prc, 
		CONVERSION_this:= downstream_backup_di_dchk_shd);

	digital_input_shadow_init(
		sim_mode:= SHADOW_SIMULATION_MODE_AUTOMATIC, 
		father:= csp_case_discharge_reject_sensors.reject_backup_di, 
		process:= dbg_root.prc, 
		CONVERSION_this:= reject_backup_di_shd);

	digital_check_shadow_init(
		sim_mode:= SHADOW_SIMULATION_MODE_AUTOMATIC, 
		father:= csp_case_discharge_reject_sensors.reject_backup_di_dchk, 
		process:= dbg_root.prc, 
		CONVERSION_this:= reject_backup_di_dchk_shd);

	digital_input_shadow_init(
		sim_mode:= SHADOW_SIMULATION_MODE_AUTOMATIC, 
		father:= csp_case_discharge_reject_sensors.reject_present_di, 
		process:= dbg_root.prc, 
		CONVERSION_this:= reject_present_di_shd);

	digital_check_shadow_init(
		sim_mode:= SHADOW_SIMULATION_MODE_AUTOMATIC, 
		father:= csp_case_discharge_reject_sensors.reject_present_di_dchk, 
		process:= dbg_root.prc, 
		CONVERSION_this:= reject_present_di_dchk_shd);

	digital_input_shadow_init(
		sim_mode:= SHADOW_SIMULATION_MODE_AUTOMATIC, 
		father:= csp_case_discharge_reject_sensors.reject_trigger_di, 
		process:= dbg_root.prc, 
		CONVERSION_this:= reject_trigger_di_shd);

	check_section_shadow_init(
		sim_mode:= SHADOW_SIMULATION_MODE_AUTOMATIC, 
		father:= csp_case_discharge_reject_sensors.reject_trigger_inchoerence_chksect, 
		process:= dbg_root.prc, 
		CONVERSION_this:= reject_trigger_inchoerence_chksect_shd);

	RETURN;
END_IF

IF	objects_running()
THEN
	digital_input_shadow_cycle(downstream_backup_di_shd);
	digital_check_shadow_cycle(downstream_backup_di_dchk_shd);
	digital_input_shadow_cycle(reject_backup_di_shd);
	digital_check_shadow_cycle(reject_backup_di_dchk_shd);
	digital_input_shadow_cycle(reject_present_di_shd);
	digital_check_shadow_cycle(reject_present_di_dchk_shd);
	digital_input_shadow_cycle(reject_trigger_di_shd);
END_IF
END_ACTION

END_PROGRAM

// ---- _Debug/dbg_csp_case_discharge_speedbelt_ls.TcPOU

(********************* G.D S.p.A. - Technical Department ***********************************
This program has been generated automatically from Application Designer DE&F
********************************************************************************************)
PROGRAM dbg_csp_case_discharge_speedbelt_ls
VAR
  axis_shd : axis_shadow;
END_VAR

_objects_manager();

IF	g_application_status <> APPLICATION_STATUS_RUNNING
THEN
	RETURN;
END_IF

CASE process_get_mode(CONVERSION_this := dbg_root.prc) OF
	MODE_ABSENT,
	MODE_INACTIVE:
		RETURN;
	MODE_TEST:
		RETURN;
END_CASE

ACTION _objects_manager:
IF	objects_initialization()
THEN
	axis_shadow_init(
		sim_mode:= SHADOW_SIMULATION_MODE_AUTOMATIC, 
		father:= csp_case_discharge_speedbelt_ls.axis, 
		process:= dbg_root.prc, 
		CONVERSION_this:= axis_shd);

	RETURN;
END_IF

IF	objects_running()
THEN
	axis_shadow_cycle(axis_shd);
END_IF
END_ACTION

END_PROGRAM

// ---- _Debug/dbg_csp_case_discharge_speedbelt_os.TcPOU

(********************* G.D S.p.A. - Technical Department ***********************************
This program has been generated automatically from Application Designer DE&F
********************************************************************************************)
PROGRAM dbg_csp_case_discharge_speedbelt_os
VAR
  axis_shd : axis_shadow;
END_VAR

_objects_manager();

IF	g_application_status <> APPLICATION_STATUS_RUNNING
THEN
	RETURN;
END_IF

CASE process_get_mode(CONVERSION_this := dbg_root.prc) OF
	MODE_ABSENT,
	MODE_INACTIVE:
		RETURN;
	MODE_TEST:
		RETURN;
END_CASE

ACTION _objects_manager:
IF	objects_initialization()
THEN
	axis_shadow_init(
		sim_mode:= SHADOW_SIMULATION_MODE_AUTOMATIC, 
		father:= csp_case_discharge_speedbelt_os.axis, 
		process:= dbg_root.prc, 
		CONVERSION_this:= axis_shd);

	RETURN;
END_IF

IF	objects_running()
THEN
	axis_shadow_cycle(axis_shd);
END_IF
END_ACTION

END_PROGRAM

// ---- _Debug/dbg_csp_case_fc_ls_lower_follower.TcPOU

(********************* G.D S.p.A. - Technical Department ***********************************
This program has been generated automatically from Application Designer DE&F
********************************************************************************************)
PROGRAM dbg_csp_case_fc_ls_lower_follower
VAR
  axis_shd : axis_shadow;
END_VAR

_objects_manager();

IF	g_application_status <> APPLICATION_STATUS_RUNNING
THEN
	RETURN;
END_IF

CASE process_get_mode(CONVERSION_this := dbg_root.prc) OF
	MODE_ABSENT,
	MODE_INACTIVE:
		RETURN;
	MODE_TEST:
		RETURN;
END_CASE

ACTION _objects_manager:
IF	objects_initialization()
THEN
	axis_shadow_init(
		sim_mode:= SHADOW_SIMULATION_MODE_AUTOMATIC, 
		father:= csp_case_fc_ls_lower_follower.axis, 
		process:= dbg_root.prc, 
		CONVERSION_this:= axis_shd);

	RETURN;
END_IF

IF	objects_running()
THEN
	axis_shadow_cycle(axis_shd);
END_IF
END_ACTION

END_PROGRAM

// ---- _Debug/dbg_csp_case_fc_ls_lower_sensors.TcPOU

(********************* G.D S.p.A. - Technical Department ***********************************
This program has been generated automatically from Application Designer DE&F
********************************************************************************************)
PROGRAM dbg_csp_case_fc_ls_lower_sensors
VAR
  flap_chksect_shd : check_section_shadow;
  flap_di_shd : digital_input_shadow;
END_VAR

_objects_manager();

IF	g_application_status <> APPLICATION_STATUS_RUNNING
THEN
	RETURN;
END_IF

CASE process_get_mode(CONVERSION_this := dbg_root.prc) OF
	MODE_ABSENT,
	MODE_INACTIVE:
		RETURN;
	MODE_TEST:
		RETURN;
END_CASE

ACTION _objects_manager:
IF	objects_initialization()
THEN
	check_section_shadow_init(
		sim_mode:= SHADOW_SIMULATION_MODE_AUTOMATIC, 
		father:= csp_case_fc_ls_lower_sensors.flap_chksect, 
		process:= dbg_root.prc, 
		CONVERSION_this:= flap_chksect_shd);

	digital_input_shadow_init(
		sim_mode:= SHADOW_SIMULATION_MODE_AUTOMATIC, 
		father:= csp_case_fc_ls_lower_sensors.flap_di, 
		process:= dbg_root.prc, 
		CONVERSION_this:= flap_di_shd);

	RETURN;
END_IF

IF	objects_running()
THEN
	digital_input_shadow_cycle(flap_di_shd);
END_IF
END_ACTION

END_PROGRAM

// ---- _Debug/dbg_csp_case_fc_ls_lower_spreader.TcPOU

(********************* G.D S.p.A. - Technical Department ***********************************
This program has been generated automatically from Application Designer DE&F
********************************************************************************************)
PROGRAM dbg_csp_case_fc_ls_lower_spreader
VAR
  axis_shd : axis_shadow;
END_VAR

_objects_manager();

IF	g_application_status <> APPLICATION_STATUS_RUNNING
THEN
	RETURN;
END_IF

CASE process_get_mode(CONVERSION_this := dbg_root.prc) OF
	MODE_ABSENT,
	MODE_INACTIVE:
		RETURN;
	MODE_TEST:
		RETURN;
END_CASE

ACTION _objects_manager:
IF	objects_initialization()
THEN
	axis_shadow_init(
		sim_mode:= SHADOW_SIMULATION_MODE_AUTOMATIC, 
		father:= csp_case_fc_ls_lower_spreader.axis, 
		process:= dbg_root.prc, 
		CONVERSION_this:= axis_shd);

	RETURN;
END_IF

IF	objects_running()
THEN
	axis_shadow_cycle(axis_shd);
END_IF
END_ACTION

END_PROGRAM

// ---- _Debug/dbg_csp_case_fc_ls_lower_trailingcloser.TcPOU

(********************* G.D S.p.A. - Technical Department ***********************************
This program has been generated automatically from Application Designer DE&F
********************************************************************************************)
PROGRAM dbg_csp_case_fc_ls_lower_trailingcloser
VAR
  axis_shd : axis_shadow;
END_VAR

_objects_manager();

IF	g_application_status <> APPLICATION_STATUS_RUNNING
THEN
	RETURN;
END_IF

CASE process_get_mode(CONVERSION_this := dbg_root.prc) OF
	MODE_ABSENT,
	MODE_INACTIVE:
		RETURN;
	MODE_TEST:
		RETURN;
END_CASE

ACTION _objects_manager:
IF	objects_initialization()
THEN
	axis_shadow_init(
		sim_mode:= SHADOW_SIMULATION_MODE_AUTOMATIC, 
		father:= csp_case_fc_ls_lower_trailingcloser.axis, 
		process:= dbg_root.prc, 
		CONVERSION_this:= axis_shd);

	RETURN;
END_IF

IF	objects_running()
THEN
	axis_shadow_cycle(axis_shd);
END_IF
END_ACTION

END_PROGRAM

// ---- _Debug/dbg_csp_case_fc_ls_upper_follower.TcPOU

(********************* G.D S.p.A. - Technical Department ***********************************
This program has been generated automatically from Application Designer DE&F
********************************************************************************************)
PROGRAM dbg_csp_case_fc_ls_upper_follower
VAR
  axis_shd : axis_shadow;
END_VAR

_objects_manager();

IF	g_application_status <> APPLICATION_STATUS_RUNNING
THEN
	RETURN;
END_IF

CASE process_get_mode(CONVERSION_this := dbg_root.prc) OF
	MODE_ABSENT,
	MODE_INACTIVE:
		RETURN;
	MODE_TEST:
		RETURN;
END_CASE

ACTION _objects_manager:
IF	objects_initialization()
THEN
	axis_shadow_init(
		sim_mode:= SHADOW_SIMULATION_MODE_AUTOMATIC, 
		father:= csp_case_fc_ls_upper_follower.axis, 
		process:= dbg_root.prc, 
		CONVERSION_this:= axis_shd);

	RETURN;
END_IF

IF	objects_running()
THEN
	axis_shadow_cycle(axis_shd);
END_IF
END_ACTION

END_PROGRAM

// ---- _Debug/dbg_csp_case_fc_ls_upper_leadingminorcloser.TcPOU

(********************* G.D S.p.A. - Technical Department ***********************************
This program has been generated automatically from Application Designer DE&F
********************************************************************************************)
PROGRAM dbg_csp_case_fc_ls_upper_leadingminorcloser
VAR
  axis_shd : axis_shadow;
END_VAR

_objects_manager();

IF	g_application_status <> APPLICATION_STATUS_RUNNING
THEN
	RETURN;
END_IF

CASE process_get_mode(CONVERSION_this := dbg_root.prc) OF
	MODE_ABSENT,
	MODE_INACTIVE:
		RETURN;
	MODE_TEST:
		RETURN;
END_CASE

ACTION _objects_manager:
IF	objects_initialization()
THEN
	axis_shadow_init(
		sim_mode:= SHADOW_SIMULATION_MODE_AUTOMATIC, 
		father:= csp_case_fc_ls_upper_leadingminorcloser.axis, 
		process:= dbg_root.prc, 
		CONVERSION_this:= axis_shd);

	RETURN;
END_IF

IF	objects_running()
THEN
	axis_shadow_cycle(axis_shd);
END_IF
END_ACTION

END_PROGRAM

// ---- _Debug/dbg_csp_case_fc_ls_upper_sensors.TcPOU

(********************* G.D S.p.A. - Technical Department ***********************************
This program has been generated automatically from Application Designer DE&F
********************************************************************************************)
PROGRAM dbg_csp_case_fc_ls_upper_sensors
VAR
  flap_chksect_shd : check_section_shadow;
  flap_di_shd : digital_input_shadow;
END_VAR

_objects_manager();

IF	g_application_status <> APPLICATION_STATUS_RUNNING
THEN
	RETURN;
END_IF

CASE process_get_mode(CONVERSION_this := dbg_root.prc) OF
	MODE_ABSENT,
	MODE_INACTIVE:
		RETURN;
	MODE_TEST:
		RETURN;
END_CASE

ACTION _objects_manager:
IF	objects_initialization()
THEN
	check_section_shadow_init(
		sim_mode:= SHADOW_SIMULATION_MODE_AUTOMATIC, 
		father:= csp_case_fc_ls_upper_sensors.flap_chksect, 
		process:= dbg_root.prc, 
		CONVERSION_this:= flap_chksect_shd);

	digital_input_shadow_init(
		sim_mode:= SHADOW_SIMULATION_MODE_AUTOMATIC, 
		father:= csp_case_fc_ls_upper_sensors.flap_di, 
		process:= dbg_root.prc, 
		CONVERSION_this:= flap_di_shd);

	RETURN;
END_IF

IF	objects_running()
THEN
	digital_input_shadow_cycle(flap_di_shd);
END_IF
END_ACTION

END_PROGRAM

// ---- _Debug/dbg_csp_case_fc_ls_upper_spreader.TcPOU

(********************* G.D S.p.A. - Technical Department ***********************************
This program has been generated automatically from Application Designer DE&F
********************************************************************************************)
PROGRAM dbg_csp_case_fc_ls_upper_spreader
VAR
  axis_shd : axis_shadow;
END_VAR

_objects_manager();

IF	g_application_status <> APPLICATION_STATUS_RUNNING
THEN
	RETURN;
END_IF

CASE process_get_mode(CONVERSION_this := dbg_root.prc) OF
	MODE_ABSENT,
	MODE_INACTIVE:
		RETURN;
	MODE_TEST:
		RETURN;
END_CASE

ACTION _objects_manager:
IF	objects_initialization()
THEN
	axis_shadow_init(
		sim_mode:= SHADOW_SIMULATION_MODE_AUTOMATIC, 
		father:= csp_case_fc_ls_upper_spreader.axis, 
		process:= dbg_root.prc, 
		CONVERSION_this:= axis_shd);

	RETURN;
END_IF

IF	objects_running()
THEN
	axis_shadow_cycle(axis_shd);
END_IF
END_ACTION

END_PROGRAM

// ---- _Debug/dbg_csp_case_fc_os_lower_follower.TcPOU

(********************* G.D S.p.A. - Technical Department ***********************************
This program has been generated automatically from Application Designer DE&F
********************************************************************************************)
PROGRAM dbg_csp_case_fc_os_lower_follower
VAR
  axis_shd : axis_shadow;
END_VAR

_objects_manager();

IF	g_application_status <> APPLICATION_STATUS_RUNNING
THEN
	RETURN;
END_IF

CASE process_get_mode(CONVERSION_this := dbg_root.prc) OF
	MODE_ABSENT,
	MODE_INACTIVE:
		RETURN;
	MODE_TEST:
		RETURN;
END_CASE

ACTION _objects_manager:
IF	objects_initialization()
THEN
	axis_shadow_init(
		sim_mode:= SHADOW_SIMULATION_MODE_AUTOMATIC, 
		father:= csp_case_fc_os_lower_follower.axis, 
		process:= dbg_root.prc, 
		CONVERSION_this:= axis_shd);

	RETURN;
END_IF

IF	objects_running()
THEN
	axis_shadow_cycle(axis_shd);
END_IF
END_ACTION

END_PROGRAM

// ---- _Debug/dbg_csp_case_fc_os_lower_sensors.TcPOU

(********************* G.D S.p.A. - Technical Department ***********************************
This program has been generated automatically from Application Designer DE&F
********************************************************************************************)
PROGRAM dbg_csp_case_fc_os_lower_sensors
VAR
  flap_chksect_shd : check_section_shadow;
  flap_di_shd : digital_input_shadow;
END_VAR

_objects_manager();

IF	g_application_status <> APPLICATION_STATUS_RUNNING
THEN
	RETURN;
END_IF

CASE process_get_mode(CONVERSION_this := dbg_root.prc) OF
	MODE_ABSENT,
	MODE_INACTIVE:
		RETURN;
	MODE_TEST:
		RETURN;
END_CASE

ACTION _objects_manager:
IF	objects_initialization()
THEN
	check_section_shadow_init(
		sim_mode:= SHADOW_SIMULATION_MODE_AUTOMATIC, 
		father:= csp_case_fc_os_lower_sensors.flap_chksect, 
		process:= dbg_root.prc, 
		CONVERSION_this:= flap_chksect_shd);

	digital_input_shadow_init(
		sim_mode:= SHADOW_SIMULATION_MODE_AUTOMATIC, 
		father:= csp_case_fc_os_lower_sensors.flap_di, 
		process:= dbg_root.prc, 
		CONVERSION_this:= flap_di_shd);

	RETURN;
END_IF

IF	objects_running()
THEN
	digital_input_shadow_cycle(flap_di_shd);
END_IF
END_ACTION

END_PROGRAM

// ---- _Debug/dbg_csp_case_fc_os_lower_spreader.TcPOU

(********************* G.D S.p.A. - Technical Department ***********************************
This program has been generated automatically from Application Designer DE&F
********************************************************************************************)
PROGRAM dbg_csp_case_fc_os_lower_spreader
VAR
  axis_shd : axis_shadow;
END_VAR

_objects_manager();

IF	g_application_status <> APPLICATION_STATUS_RUNNING
THEN
	RETURN;
END_IF

CASE process_get_mode(CONVERSION_this := dbg_root.prc) OF
	MODE_ABSENT,
	MODE_INACTIVE:
		RETURN;
	MODE_TEST:
		RETURN;
END_CASE

ACTION _objects_manager:
IF	objects_initialization()
THEN
	axis_shadow_init(
		sim_mode:= SHADOW_SIMULATION_MODE_AUTOMATIC, 
		father:= csp_case_fc_os_lower_spreader.axis, 
		process:= dbg_root.prc, 
		CONVERSION_this:= axis_shd);

	RETURN;
END_IF

IF	objects_running()
THEN
	axis_shadow_cycle(axis_shd);
END_IF
END_ACTION

END_PROGRAM

// ---- _Debug/dbg_csp_case_fc_os_lower_trailingcloser.TcPOU

(********************* G.D S.p.A. - Technical Department ***********************************
This program has been generated automatically from Application Designer DE&F
********************************************************************************************)
PROGRAM dbg_csp_case_fc_os_lower_trailingcloser
VAR
  axis_shd : axis_shadow;
END_VAR

_objects_manager();

IF	g_application_status <> APPLICATION_STATUS_RUNNING
THEN
	RETURN;
END_IF

CASE process_get_mode(CONVERSION_this := dbg_root.prc) OF
	MODE_ABSENT,
	MODE_INACTIVE:
		RETURN;
	MODE_TEST:
		RETURN;
END_CASE

ACTION _objects_manager:
IF	objects_initialization()
THEN
	axis_shadow_init(
		sim_mode:= SHADOW_SIMULATION_MODE_AUTOMATIC, 
		father:= csp_case_fc_os_lower_trailingcloser.axis, 
		process:= dbg_root.prc, 
		CONVERSION_this:= axis_shd);

	RETURN;
END_IF

IF	objects_running()
THEN
	axis_shadow_cycle(axis_shd);
END_IF
END_ACTION

END_PROGRAM

// ---- _Debug/dbg_csp_case_fc_os_upper_follower.TcPOU

(********************* G.D S.p.A. - Technical Department ***********************************
This program has been generated automatically from Application Designer DE&F
********************************************************************************************)
PROGRAM dbg_csp_case_fc_os_upper_follower
VAR
  axis_shd : axis_shadow;
END_VAR

_objects_manager();

IF	g_application_status <> APPLICATION_STATUS_RUNNING
THEN
	RETURN;
END_IF

CASE process_get_mode(CONVERSION_this := dbg_root.prc) OF
	MODE_ABSENT,
	MODE_INACTIVE:
		RETURN;
	MODE_TEST:
		RETURN;
END_CASE

ACTION _objects_manager:
IF	objects_initialization()
THEN
	axis_shadow_init(
		sim_mode:= SHADOW_SIMULATION_MODE_AUTOMATIC, 
		father:= csp_case_fc_os_upper_follower.axis, 
		process:= dbg_root.prc, 
		CONVERSION_this:= axis_shd);

	RETURN;
END_IF

IF	objects_running()
THEN
	axis_shadow_cycle(axis_shd);
END_IF
END_ACTION

END_PROGRAM

// ---- _Debug/dbg_csp_case_fc_os_upper_sensors.TcPOU

(********************* G.D S.p.A. - Technical Department ***********************************
This program has been generated automatically from Application Designer DE&F
********************************************************************************************)
PROGRAM dbg_csp_case_fc_os_upper_sensors
VAR
  flap_chksect_shd : check_section_shadow;
  flap_di_shd : digital_input_shadow;
END_VAR

_objects_manager();

IF	g_application_status <> APPLICATION_STATUS_RUNNING
THEN
	RETURN;
END_IF

CASE process_get_mode(CONVERSION_this := dbg_root.prc) OF
	MODE_ABSENT,
	MODE_INACTIVE:
		RETURN;
	MODE_TEST:
		RETURN;
END_CASE

ACTION _objects_manager:
IF	objects_initialization()
THEN
	check_section_shadow_init(
		sim_mode:= SHADOW_SIMULATION_MODE_AUTOMATIC, 
		father:= csp_case_fc_os_upper_sensors.flap_chksect, 
		process:= dbg_root.prc, 
		CONVERSION_this:= flap_chksect_shd);

	digital_input_shadow_init(
		sim_mode:= SHADOW_SIMULATION_MODE_AUTOMATIC, 
		father:= csp_case_fc_os_upper_sensors.flap_di, 
		process:= dbg_root.prc, 
		CONVERSION_this:= flap_di_shd);

	RETURN;
END_IF

IF	objects_running()
THEN
	digital_input_shadow_cycle(flap_di_shd);
END_IF
END_ACTION

END_PROGRAM

// ---- _Debug/dbg_csp_case_fc_os_upper_spreader.TcPOU

(********************* G.D S.p.A. - Technical Department ***********************************
This program has been generated automatically from Application Designer DE&F
********************************************************************************************)
PROGRAM dbg_csp_case_fc_os_upper_spreader
VAR
  axis_shd : axis_shadow;
END_VAR

_objects_manager();

IF	g_application_status <> APPLICATION_STATUS_RUNNING
THEN
	RETURN;
END_IF

CASE process_get_mode(CONVERSION_this := dbg_root.prc) OF
	MODE_ABSENT,
	MODE_INACTIVE:
		RETURN;
	MODE_TEST:
		RETURN;
END_CASE

ACTION _objects_manager:
IF	objects_initialization()
THEN
	axis_shadow_init(
		sim_mode:= SHADOW_SIMULATION_MODE_AUTOMATIC, 
		father:= csp_case_fc_os_upper_spreader.axis, 
		process:= dbg_root.prc, 
		CONVERSION_this:= axis_shd);

	RETURN;
END_IF

IF	objects_running()
THEN
	axis_shadow_cycle(axis_shd);
END_IF
END_ACTION

END_PROGRAM

// ---- _Debug/dbg_csp_case_feed_arm_elbow.TcPOU

(********************* G.D S.p.A. - Technical Department ***********************************
This program has been generated automatically from Application Designer DE&F
********************************************************************************************)
PROGRAM dbg_csp_case_feed_arm_elbow
VAR
  axis_shd : axis_shadow;
END_VAR

_objects_manager();

IF	g_application_status <> APPLICATION_STATUS_RUNNING
THEN
	RETURN;
END_IF

CASE process_get_mode(CONVERSION_this := dbg_root.prc) OF
	MODE_ABSENT,
	MODE_INACTIVE:
		RETURN;
	MODE_TEST:
		RETURN;
END_CASE

ACTION _objects_manager:
IF	objects_initialization()
THEN
	axis_shadow_init(
		sim_mode:= SHADOW_SIMULATION_MODE_AUTOMATIC, 
		father:= csp_case_feed_arm_elbow.axis, 
		process:= dbg_root.prc, 
		CONVERSION_this:= axis_shd);

	RETURN;
END_IF

IF	objects_running()
THEN
	axis_shadow_cycle(axis_shd);
END_IF
END_ACTION

END_PROGRAM

// ---- _Debug/dbg_csp_case_feed_arm_sensors.TcPOU

(********************* G.D S.p.A. - Technical Department ***********************************
This program has been generated automatically from Application Designer DE&F
********************************************************************************************)
PROGRAM dbg_csp_case_feed_arm_sensors
VAR
  case_check_chksect_shd : check_section_shadow;
  case_check_di_shd : digital_input_shadow;
  case_check_inchoerence_chksect_shd : check_section_shadow;
  major_vacuum_do_shd : digital_output_shadow;
  major_vacuum_sact_shd : digital_actuator_shadow;
  minor_vacuum_do_shd : digital_output_shadow;
  minor_vacuum_sact_shd : digital_actuator_shadow;
END_VAR

_objects_manager();

IF	g_application_status <> APPLICATION_STATUS_RUNNING
THEN
	RETURN;
END_IF

CASE process_get_mode(CONVERSION_this := dbg_root.prc) OF
	MODE_ABSENT,
	MODE_INACTIVE:
		RETURN;
	MODE_TEST:
		RETURN;
END_CASE

ACTION _objects_manager:
IF	objects_initialization()
THEN

	digital_input_shadow_init(
		sim_mode:= SHADOW_SIMULATION_MODE_AUTOMATIC, 
		father:= csp_case_feed_arm_sensors.case_check_di, 
		process:= dbg_root.prc, 
		CONVERSION_this:= case_check_di_shd);

	check_section_shadow_init(
		sim_mode:= SHADOW_SIMULATION_MODE_AUTOMATIC, 
		father:= csp_case_feed_arm_sensors.case_check_inchoerence_chksect, 
		process:= dbg_root.prc, 
		CONVERSION_this:= case_check_inchoerence_chksect_shd);

	digital_output_shadow_init(
		sim_mode:= SHADOW_SIMULATION_MODE_AUTOMATIC, 
		father:= csp_case_feed_arm_sensors.major_vacuum_do, 
		process:= dbg_root.prc, 
		CONVERSION_this:= major_vacuum_do_shd);

	digital_actuator_shadow_init(
		sim_mode:= SHADOW_SIMULATION_MODE_AUTOMATIC, 
		father:= csp_case_feed_arm_sensors.major_vacuum_sact, 
		process:= dbg_root.prc, 
		CONVERSION_this:= major_vacuum_sact_shd);

	digital_output_shadow_init(
		sim_mode:= SHADOW_SIMULATION_MODE_AUTOMATIC, 
		father:= csp_case_feed_arm_sensors.minor_vacuum_do, 
		process:= dbg_root.prc, 
		CONVERSION_this:= minor_vacuum_do_shd);

	digital_actuator_shadow_init(
		sim_mode:= SHADOW_SIMULATION_MODE_AUTOMATIC, 
		father:= csp_case_feed_arm_sensors.minor_vacuum_sact, 
		process:= dbg_root.prc, 
		CONVERSION_this:= minor_vacuum_sact_shd);

	RETURN;
END_IF

IF	objects_running()
THEN
	digital_input_shadow_cycle(case_check_di_shd);
	digital_output_shadow_cycle(major_vacuum_do_shd);
	digital_actuator_shadow_cycle(major_vacuum_sact_shd);
	digital_output_shadow_cycle(minor_vacuum_do_shd);
	digital_actuator_shadow_cycle(minor_vacuum_sact_shd);
END_IF
END_ACTION

END_PROGRAM

// ---- _Debug/dbg_csp_case_feed_arm_shoulder.TcPOU

(********************* G.D S.p.A. - Technical Department ***********************************
This program has been generated automatically from Application Designer DE&F
********************************************************************************************)
PROGRAM dbg_csp_case_feed_arm_shoulder
VAR
  axis_shd : axis_shadow;
END_VAR

_objects_manager();

IF	g_application_status <> APPLICATION_STATUS_RUNNING
THEN
	RETURN;
END_IF

CASE process_get_mode(CONVERSION_this := dbg_root.prc) OF
	MODE_ABSENT,
	MODE_INACTIVE:
		RETURN;
	MODE_TEST:
		RETURN;
END_CASE

ACTION _objects_manager:
IF	objects_initialization()
THEN
	axis_shadow_init(
		sim_mode:= SHADOW_SIMULATION_MODE_AUTOMATIC, 
		father:= csp_case_feed_arm_shoulder.axis, 
		process:= dbg_root.prc, 
		CONVERSION_this:= axis_shd);

	RETURN;
END_IF

IF	objects_running()
THEN
	axis_shadow_cycle(axis_shd);
END_IF
END_ACTION

END_PROGRAM

// ---- _Debug/dbg_csp_case_feed_arm_wrist.TcPOU

(********************* G.D S.p.A. - Technical Department ***********************************
This program has been generated automatically from Application Designer DE&F
********************************************************************************************)
PROGRAM dbg_csp_case_feed_arm_wrist
VAR
  axis_shd : axis_shadow;
END_VAR

_objects_manager();

IF	g_application_status <> APPLICATION_STATUS_RUNNING
THEN
	RETURN;
END_IF

CASE process_get_mode(CONVERSION_this := dbg_root.prc) OF
	MODE_ABSENT,
	MODE_INACTIVE:
		RETURN;
	MODE_TEST:
		RETURN;
END_CASE

ACTION _objects_manager:
IF	objects_initialization()
THEN
	axis_shadow_init(
		sim_mode:= SHADOW_SIMULATION_MODE_AUTOMATIC, 
		father:= csp_case_feed_arm_wrist.axis, 
		process:= dbg_root.prc, 
		CONVERSION_this:= axis_shd);

	RETURN;
END_IF

IF	objects_running()
THEN
	axis_shadow_cycle(axis_shd);
END_IF
END_ACTION

END_PROGRAM

// ---- _Debug/dbg_csp_case_feed_kinematic_tilt.TcPOU

(********************* G.D S.p.A. - Technical Department ***********************************
This program has been generated automatically from Application Designer DE&F
********************************************************************************************)
PROGRAM dbg_csp_case_feed_kinematic_tilt
VAR
  axis_shd : axis_shadow;
END_VAR

_objects_manager();

IF	g_application_status <> APPLICATION_STATUS_RUNNING
THEN
	RETURN;
END_IF

CASE process_get_mode(CONVERSION_this := dbg_root.prc) OF
	MODE_ABSENT,
	MODE_INACTIVE:
		RETURN;
	MODE_TEST:
		RETURN;
END_CASE

ACTION _objects_manager:
IF	objects_initialization()
THEN
	axis_shadow_init(
		sim_mode:= SHADOW_SIMULATION_MODE_AUTOMATIC, 
		father:= csp_case_feed_kinematic_tilt.axis, 
		process:= dbg_root.prc, 
		CONVERSION_this:= axis_shd);

	RETURN;
END_IF

IF	objects_running()
THEN
	axis_shadow_cycle(axis_shd);
END_IF
END_ACTION

END_PROGRAM

// ---- _Debug/dbg_csp_case_feed_kinematic_x.TcPOU

(********************* G.D S.p.A. - Technical Department ***********************************
This program has been generated automatically from Application Designer DE&F
********************************************************************************************)
PROGRAM dbg_csp_case_feed_kinematic_x
VAR
  axis_shd : axis_shadow;
END_VAR

_objects_manager();

IF	g_application_status <> APPLICATION_STATUS_RUNNING
THEN
	RETURN;
END_IF

CASE process_get_mode(CONVERSION_this := dbg_root.prc) OF
	MODE_ABSENT,
	MODE_INACTIVE:
		RETURN;
	MODE_TEST:
		RETURN;
END_CASE

ACTION _objects_manager:
IF	objects_initialization()
THEN
	axis_shadow_init(
		sim_mode:= SHADOW_SIMULATION_MODE_AUTOMATIC, 
		father:= csp_case_feed_kinematic_x.axis, 
		process:= dbg_root.prc, 
		CONVERSION_this:= axis_shd);

	RETURN;
END_IF

IF	objects_running()
THEN
	axis_shadow_cycle(axis_shd);
END_IF
END_ACTION

END_PROGRAM

// ---- _Debug/dbg_csp_case_feed_kinematic_y.TcPOU

(********************* G.D S.p.A. - Technical Department ***********************************
This program has been generated automatically from Application Designer DE&F
********************************************************************************************)
PROGRAM dbg_csp_case_feed_kinematic_y
VAR
  axis_shd : axis_shadow;
END_VAR

_objects_manager();

IF	g_application_status <> APPLICATION_STATUS_RUNNING
THEN
	RETURN;
END_IF

CASE process_get_mode(CONVERSION_this := dbg_root.prc) OF
	MODE_ABSENT,
	MODE_INACTIVE:
		RETURN;
	MODE_TEST:
		RETURN;
END_CASE

ACTION _objects_manager:
IF	objects_initialization()
THEN
	axis_shadow_init(
		sim_mode:= SHADOW_SIMULATION_MODE_AUTOMATIC, 
		father:= csp_case_feed_kinematic_y.axis, 
		process:= dbg_root.prc, 
		CONVERSION_this:= axis_shd);

	RETURN;
END_IF

IF	objects_running()
THEN
	axis_shadow_cycle(axis_shd);
END_IF
END_ACTION

END_PROGRAM

// ---- _Debug/dbg_csp_case_feed_magazine_accu_lsdepth.TcPOU

(********************* G.D S.p.A. - Technical Department ***********************************
This program has been generated automatically from Application Designer DE&F
********************************************************************************************)
PROGRAM dbg_csp_case_feed_magazine_accu_lsdepth
VAR
  axis_shd : axis_shadow;
END_VAR

_objects_manager();

IF	g_application_status <> APPLICATION_STATUS_RUNNING
THEN
	RETURN;
END_IF

CASE process_get_mode(CONVERSION_this := dbg_root.prc) OF
	MODE_ABSENT,
	MODE_INACTIVE:
		RETURN;
	MODE_TEST:
		RETURN;
END_CASE

ACTION _objects_manager:
IF	objects_initialization()
THEN
	axis_shadow_init(
		sim_mode:= SHADOW_SIMULATION_MODE_AUTOMATIC, 
		father:= csp_case_feed_magazine_accu_lsdepth.axis, 
		process:= dbg_root.prc, 
		CONVERSION_this:= axis_shd);

	RETURN;
END_IF

IF	objects_running()
THEN
	axis_shadow_cycle(axis_shd);
END_IF
END_ACTION

END_PROGRAM

// ---- _Debug/dbg_csp_case_feed_magazine_accu_osdepth.TcPOU

